// TIA Portal project "KNX_SPS_Forum_Van" (V18)

(* hardware
DEVICE "S7-1200-Station_1"  S7-1200 Station
   slot 0: "Baugruppenträger_0"  S7-1200 Rack  Rack  V1.0
   slot 1: "PLC_1"  CPU 1214C DC/DC/DC  6ES7 214-1AG40-0XB0  V4.6
*)

// ===== PLC "PLC_1"  CPU 1214C DC/DC/DC =====

VAR_GLOBAL CONSTANT   // PLC tag table "CONST_KNX"
   "KNX_ARRAY_MAX" : Int := 49;
END_VAR

VAR_GLOBAL CONSTANT   // PLC tag table "CONST_Ethernet"
   "CONN_ID_KNX" : Int := 1;
   "CONN_ID_SMA" : Conn_Ouc := 2;
   "CONN_ID_RASENROBI" : Conn_Ouc := 3;
   "CONN_ID_VOLKSZAEHLER_GET" : Conn_Ouc := 4;
   "CONN_ID_SHELLY" : Conn_Ouc := 5;
   "CONN_ID_VOLKSZAEHLER_POST" : Conn_Ouc := 6;
   "CONN_ID_WALLBOX" : Conn_Ouc := 7;
   "CONN_ID_Res8" : Conn_Ouc := 8;
   "Maximal 8 OU Verbindungen" : Conn_Ouc := 8888;   // Maximal 8 OU Verbindungen
END_VAR

// folder: KNX

TYPE "KNX_Data_Exchange"
   STRUCT
      Empf_Dat : "KNX_Empf_Dat";
      Send_Dat : "KNX_Send_Dat";
      Senden : Bool;
      Empfangen : Bool;
   END_STRUCT;
   // // Empf_Dat.Daten[1] : APCI + 6Bit Nutzdaten
END_TYPE

TYPE "KNX_Empf_Dat"
   STRUCT
      GruppenAddr : Word;
      Laenge : Byte;
      NPDU_ABCI : Byte;
      Daten : Array[1..20] of Byte;
   END_STRUCT;
END_TYPE

TYPE "KNX_Send_Dat"
   STRUCT
      GruppenAddr : Word;
      Laenge : Byte;
      NPDU_ABCI : Byte;
      Daten : Array[1..20] of Byte;
   END_STRUCT;
END_TYPE

TYPE "KNX_Data_Exchange_bak"
   STRUCT
      Empf_Dat : Struct
         GruppenAddr : Word;
         Laenge : Byte;
         NPDU_ABCI : Byte;
         Daten : Array[1..20] of Byte;
      END_STRUCT;
      Send_Dat : Struct
         GruppenAddr : Word;
         Laenge : Byte;
         NPDU_ABCI : Byte;
         Daten : Array[1..20] of Byte;
      END_STRUCT;
      Senden : Bool;
      Empfangen : Bool;
   END_STRUCT;
END_TYPE

TYPE "KNX_GA_Nr"
   STRUCT
      haupt : USInt;   // Hauptgruppe = 0..31
      mittel : USInt;   // Mittelgruppe = 0..7
      unter : USInt;   // Untergruppe = 0..255
   END_STRUCT;
END_TYPE

TYPE "KNX_Log_empf"
   STRUCT
      ga_nr : "KNX_GA_Nr";
      Empf_Dat : "KNX_Empf_Dat";
   END_STRUCT;
END_TYPE

TYPE "KNX_test_2"
   STRUCT
      GA : "KNX_GA_Nr";
      para : Struct
         aktiv : Bool;
         abfragbar : Bool;   // ReadRequest vom(!) Bus beantworten
         beschreibbar : Bool;   // Write vom(!) Bus zulassen
         initScan : Bool;   // ist diese Option aktiviert wird der KO-Wert beim Start vom KNX-Bus abgefragt (Read-Request)
         sendByChange : Bool;
         sendByChangeValue : Real;
      END_STRUCT;
      cmd : Struct
         send : Bool;   // SPS Wert an den Bus senden
         sendReadRequest : Bool;   // Wert vom Bus abfragen
      END_STRUCT;
      value : Struct
         DPT : UInt;
         DPT1 : Bool;
         DPT2 : Byte;
         DPT3 : Byte;
         DPT4 : Char;
         DPT5 : USInt;
         DPT6 : SInt;
         DPT7 : UInt;
         DPT8 : Int;
         DPT9 : Real;
         DPT10x : Bool;
         DPT11x : Bool;
         DPT12 : UDInt;
         DPT13 : DInt;
         DPT14 : Real;
      END_STRUCT;
   END_STRUCT;
END_TYPE

TYPE "KNX_test_1"
   STRUCT
      GA : "KNX_GA_Nr";
      para : Struct
         aktiv : Bool;
         abfragbar : Bool;   // ReadRequest vom(!) Bus beantworten
         beschreibbar : Bool;   // Write vom(!) Bus zulassen
         initScan : Bool;   // ist diese Option aktiviert wird der KO-Wert beim Start vom KNX-Bus abgefragt (Read-Request)
         sendByChange : Bool;
         sendByChangeValue : Real;
      END_STRUCT;
      cmd : Struct
         send : Bool;   // SPS Wert an den Bus senden
         sendReadRequest : Bool;   // Wert vom Bus abfragen
      END_STRUCT;
      value : Struct
         DPT : Int;
         raw : Array[0..14] of Byte;
      END_STRUCT;
   END_STRUCT;
END_TYPE

TYPE "KNX_KO"
   STRUCT
      GA : "KNX_GA_Nr";   // Gruppenadresse
      para : Struct   // Parameter
         aktiv : Bool;   // KO ist aktiv und wird bearbeitet
         abfragbarVomBus : Bool;   // SPS Sendet Wert auf den Bus - ReadRequest vom(!) Bus beantworten
         beschreibbarVomBus : Bool;   // SPS empfängt Wert vom Bus - Write vom(!) Bus zulassen
         initScan : Bool;   // ist diese Option aktiviert wird der KO-Wert beim Start vom KNX-Bus abgefragt (Read-Request)
         sendByChange : Bool;   // Auf den Bus senden wenn sich der SPS Wert geändert hat
         sendByChangeValue : Real;   // diffferenz um den sich der Wert ändern muss
      END_STRUCT;
      cmd : Struct   // Kommando
         send : Bool;   // SPS Wert an den Bus senden
         readRequest : Bool;   // Wert vom Bus abfragen
      END_STRUCT;
      stat : Struct   // Status
         newTelegramRec : Bool;   // Neues Telegram empfangen
         newTelegramSend : Bool;   // Telegram gesendet
         counterRec : UInt;   // Zähler Telegramme Empfangen (Flanke)
         counterSend : UInt;   // Zähler Telegramme Gesendet
      END_STRUCT;
   END_STRUCT;
END_TYPE

TYPE "KNX_DPT3"
   STRUCT
      Down_Increase : Bool;   // 0 = Up, Decrease / 1 = Down, Increase
      prozent : USInt;   // 1, 3, 6, 12, 25, 50, 100% / 0 = Stopp
   END_STRUCT;
END_TYPE

// folder: 10 Haus Logik/instanzen

DATA_BLOCK "aussen-rasenrobi_DB"   // DB8
{ S7_Optimized_Access := 'TRUE' }
VERSION : 0.1
// stored: InstanceOfName aussen-rasenrobi
"aussen-rasenrobi"
BEGIN
END_DATA_BLOCK

DATA_BLOCK "eg-Wohn-Ess-Kueche_DB"   // DB17
{ S7_Optimized_Access := 'TRUE' }
VERSION : 0.1
// stored: InstanceOfName eg-Wohn-Ess-Kueche
"eg-Wohn-Ess-Kueche"
BEGIN
END_DATA_BLOCK

DATA_BLOCK "zental-strom_DB"   // DB21
{ S7_Optimized_Access := 'TRUE' }
VERSION : 0.1
// stored: InstanceOfName zental-strom
"zental-strom"
BEGIN
END_DATA_BLOCK

DATA_BLOCK "zentral-wasser_DB"   // DB33
{ S7_Optimized_Access := 'TRUE' }
VERSION : 0.1
// stored: InstanceOfName zentral-wasser
"zentral-wasser"
BEGIN
END_DATA_BLOCK

DATA_BLOCK "zentral-beschattung_DB"   // DB35
{ S7_Optimized_Access := 'TRUE' }
VERSION : 0.1
// stored: InstanceOfName zentral-beschattung
"zentral-beschattung"
BEGIN
END_DATA_BLOCK

// folder: 20 KNX

DATA_BLOCK "db-knx-Allg"   // DB2
{ S7_Optimized_Access := 'TRUE' }
VERSION : 0.1
   VAR
      "Disconnect Count" : Int;
      DisconnectChannelID : Array[1..20] of Byte;
      knxComOk : Bool;
      knxComTimeOut : Bool;
      initScanDone : Bool;
      knxBereit : Bool;
   END_VAR
BEGIN
END_DATA_BLOCK

DATA_BLOCK "db-knx-log"   // DB4
{ S7_Optimized_Access := 'TRUE' }
VERSION : 0.1
   VAR
      index : Int;
      empf : Array[0..100] of "KNX_Log_empf";
   END_VAR
BEGIN
END_DATA_BLOCK

DATA_BLOCK "db-knx-com"   // DB10
{ S7_Optimized_Access := 'TRUE' }
VERSION : 0.1
   VAR
      KNXDat : "KNX_Data_Exchange";   // KNX: Datenaustausch zwischen den FBs
   END_VAR
BEGIN
END_DATA_BLOCK

DATA_BLOCK "db-knx-ko"   // DB15
{ S7_Optimized_Access := 'TRUE' }
VERSION : 0.1
   VAR
      ko : Array[0.."KNX_ARRAY_MAX"] of "KNX_KO";   // Kommunikationsobjekt
      koVal : Struct   // Kommunikationsobjekt Wert
         "0_Terassen-Tür (Zu=Aus=0 / Auf=Ein=1)" : Bool;   // 6/1/2 = Terassen-Tür (Zu=Aus=0 / Auf=Ein=1)
         "1_Wohn-Ess-Kueche.Terasse(Patch-kurz)" : Bool;   // 6/1/6 = Wohn-Ess-Kueche.Terasse(Patch-kurz)
         "2_Wohn-Ess-Küche.Szene" : USInt;   // 8/1/1 = Wohn-Ess-Küche.Szene
         "3_Wohnen-Tür-SW.Jal(Jalousie Auf/Ab)" : Bool;   // 3/1/140 = Wohnen-Tür-SW.Jal(Jalousie Auf/Ab)
         "4_Zisterne(Fuellstand qm)" : Real;   // 6/3/140 = Zisterne(Fuellstand qm)
         "5_PV-Anlage(Erzeugung)" : Real;   // 6/3/141 = PV-Anlage(Erzeugung) / DPT 9.024 Leistung (kW)
         "6_Stromzaehler(In-Out-Aktuell)" : Real;   // 6/0/0 = Stromzaehler(In-Out-Aktuell) / Positiv=Bezug vom Netz / Negativ = Verkauf an Netz / / DPT 9.024 Leistung (kW)
         "7_Strom(Eigenverbrauch)" : Real;   // 6/0/1 = Strom(Eigenverbrauch) / DPT 9.024 Leistung (kW)
         "8_Zirkulation.WarmWasser(Ein)" : Bool;   // 7/0/1 = Zirkulation.WarmWasser(Ein)
         "9_Umwelt.Wetterstation(Helligkeit O Messwert)" : Real;   // 6/3/0 = Umwelt.Wetterstation(Helligkeit O Messwert)
         "10_Umwelt.Wetterstation(Helligkeit S Messwert)" : Real;   // 6/3/17 = Umwelt.Wetterstation(Helligkeit S Messwert)
         "11_Umwelt.Wetterstation(Helligkeit W Messwert)" : Real;   // 6/3/34 = Umwelt.Wetterstation(Helligkeit W Messwert)
         "12_Umwelt-Garage.Lichtsensor(Helligkeit Messwert)" : Real;   // 6/3/105 = Umwelt-Garage.Lichtsensor(Helligkeit Messwert)
         "13_Beschattung(Diag)" : String[14];   // 3/1/221 = Beschattung(Diag)
         "14_Umwelt.Wetterstation(Wind Geschwindigkeit)" : Real;   // 6/3/54 = Umwelt.Wetterstation(Wind Geschwindigkeit)
         "15_Umwelt.Wetterstation(Temperatur Messwert)" : Real;   // 6/3/55 = Umwelt.Wetterstation(Temperatur Messwert)
         "16_Umwelt.Helligkeit.Max(Helligkeit)" : Real;   // 6/3/106 = Umwelt.Helligkeit.Max(Helligkeit)
         "17_Umwelt.Regensensor(Meldung Regen ja/nein)" : Bool;   // 6/3/100 = Umwelt.Regensensor(Meldung Regen ja/nein)
         "18_DPT3_Test" : "KNX_DPT3";   // 11/0/10 = DPT3 Test
      END_STRUCT;
   END_VAR
   VAR RETAIN
      initScan_nachDbReinit : Bool := false;   // Löst einen InitScan aus nachdem der DB reinitialisiert wurde
   END_VAR
BEGIN
   ko[0].GA.haupt := 6;
   ko[0].GA.mittel := 1;
   ko[0].GA.unter := 2;
   ko[0].para.aktiv := true;
   ko[0].para.abfragbarVomBus := false;
   ko[0].para.beschreibbarVomBus := true;
   ko[0].para.initScan := true;
   ko[1].GA.haupt := 6;
   ko[1].GA.mittel := 1;
   ko[1].GA.unter := 6;
   ko[1].para.aktiv := true;
   ko[1].para.abfragbarVomBus := false;
   ko[1].para.beschreibbarVomBus := true;
   ko[1].para.initScan := false;
   ko[1].para.sendByChange := false;
   ko[2].GA.haupt := 8;
   ko[2].GA.mittel := 1;
   ko[2].GA.unter := 1;
   ko[2].para.aktiv := true;
   ko[2].para.abfragbarVomBus := false;
   ko[2].para.beschreibbarVomBus := true;
   ko[2].para.initScan := false;
   ko[2].para.sendByChange := false;
   ko[3].GA.haupt := 3;
   ko[3].GA.mittel := 1;
   ko[3].GA.unter := 140;
   ko[3].para.aktiv := true;
   ko[3].para.abfragbarVomBus := false;
   ko[3].para.beschreibbarVomBus := false;
   ko[3].para.initScan := false;
   ko[4].GA.haupt := 6;
   ko[4].GA.mittel := 3;
   ko[4].GA.unter := 140;
   ko[4].para.aktiv := true;
   ko[4].para.abfragbarVomBus := true;
   ko[4].para.beschreibbarVomBus := false;
   ko[4].para.initScan := false;
   ko[4].para.sendByChange := true;
   ko[4].para.sendByChangeValue := 0.05;
   ko[5].GA.haupt := 6;
   ko[5].GA.mittel := 3;
   ko[5].GA.unter := 141;
   ko[5].para.aktiv := true;
   ko[5].para.abfragbarVomBus := true;
   ko[5].para.beschreibbarVomBus := false;
   ko[5].para.initScan := false;
   ko[5].para.sendByChange := true;
   ko[5].para.sendByChangeValue := 0.2;
   ko[6].GA.haupt := 6;
   ko[6].GA.unter := 0;
   ko[6].para.aktiv := true;
   ko[6].para.initScan := false;
   ko[7].GA.haupt := 6;
   ko[7].GA.mittel := 0;
   ko[7].GA.unter := 1;
   ko[7].para.aktiv := true;
   ko[7].para.initScan := false;
   ko[8].GA.haupt := 7;
   ko[8].GA.unter := 1;
   ko[8].para.aktiv := true;
   ko[8].GA.mittel := 0;
   ko[6].GA.mittel := 0;
   ko[6].para.abfragbarVomBus := true;
   ko[6].para.beschreibbarVomBus := false;
   ko[6].para.sendByChange := true;
   ko[6].para.sendByChangeValue := 0.2;
   ko[7].para.abfragbarVomBus := true;
   ko[7].para.beschreibbarVomBus := false;
   ko[7].para.sendByChange := true;
   ko[7].para.sendByChangeValue := 0.2;
   ko[9].GA.haupt := 6;
   ko[9].GA.mittel := 3;
   ko[9].GA.unter := 0;
   ko[9].para.aktiv := true;
   ko[9].para.abfragbarVomBus := false;
   ko[9].para.initScan := true;
   ko[9].para.beschreibbarVomBus := true;
   ko[9].para.sendByChange := false;
   ko[10].GA.haupt := 6;
   ko[10].GA.mittel := 3;
   ko[10].GA.unter := 17;
   ko[10].para.aktiv := true;
   ko[10].para.abfragbarVomBus := false;
   ko[10].para.beschreibbarVomBus := true;
   ko[10].para.initScan := true;
   ko[10].para.sendByChange := false;
   ko[11].GA.haupt := 6;
   ko[11].GA.mittel := 3;
   ko[11].GA.unter := 34;
   ko[11].para.aktiv := true;
   ko[11].para.abfragbarVomBus := false;
   ko[11].para.beschreibbarVomBus := true;
   ko[11].para.initScan := true;
   ko[11].para.sendByChange := false;
   ko[12].GA.haupt := 6;
   ko[12].GA.mittel := 3;
   ko[12].GA.unter := 105;
   ko[12].para.aktiv := true;
   ko[12].para.abfragbarVomBus := false;
   ko[12].para.beschreibbarVomBus := true;
   ko[12].para.initScan := true;
   ko[12].para.sendByChange := false;
   ko[13].GA.haupt := 3;
   ko[13].GA.mittel := 1;
   ko[13].GA.unter := 221;
   ko[13].para.aktiv := true;
   ko[13].para.abfragbarVomBus := false;
   ko[13].para.beschreibbarVomBus := true;
   ko[13].para.initScan := true;
   ko[13].para.sendByChange := false;
   ko[14].GA.haupt := 6;
   ko[14].GA.mittel := 3;
   ko[14].GA.unter := 54;
   ko[14].para.aktiv := true;
   ko[14].para.abfragbarVomBus := false;
   ko[14].para.beschreibbarVomBus := true;
   ko[14].para.initScan := true;
   ko[14].para.sendByChange := false;
   ko[15].GA.haupt := 6;
   ko[15].GA.mittel := 3;
   ko[15].GA.unter := 55;
   ko[15].para.aktiv := true;
   ko[15].para.abfragbarVomBus := false;
   ko[15].para.beschreibbarVomBus := true;
   ko[15].para.initScan := true;
   ko[15].para.sendByChange := false;
   ko[16].GA.haupt := 6;
   ko[16].GA.mittel := 3;
   ko[16].GA.unter := 106;
   ko[16].para.aktiv := true;
   ko[16].para.abfragbarVomBus := true;
   ko[16].para.beschreibbarVomBus := false;
   ko[16].para.initScan := false;
   ko[16].para.sendByChange := true;
   ko[16].para.sendByChangeValue := 100.0;
   ko[17].GA.haupt := 6;
   ko[17].GA.mittel := 3;
   ko[17].GA.unter := 100;
   ko[17].para.aktiv := true;
   ko[17].para.initScan := true;
   ko[17].para.beschreibbarVomBus := true;
   ko[18].GA.haupt := 11;
   ko[18].GA.mittel := 0;
   ko[18].GA.unter := 10;
   ko[18].para.aktiv := true;
   ko[18].para.abfragbarVomBus := true;
   ko[18].para.beschreibbarVomBus := true;
   ko[18].para.initScan := true;
   ko[18].para.sendByChange := true;
   // ko[0] : 6/1/2 = Terassen-Tür (Zu=Aus=0 / Auf=Ein=1)
   // ko[1] : 6/1/6 = Wohn-Ess-Kueche.Terasse(Patch-kurz)
   // ko[2] : 8/1/1 = Wohn-Ess-Küche.Szene
   // ko[3] : 3/1/140 = Wohnen-Tür-SW.Jal(Jalousie Auf/Ab)
   // ko[4] : 6/3/140 = Zisterne(Fuellstand qm)
   // ko[5] : 6/3/141 = PV-Anlage(Erzeugung)
   // ko[6] : 6/0/0 = Stromzaehler(In-Out-Aktuell)
   // ko[7] : 6/0/1 = Strom(Eigenverbrauch)
   // ko[8] : 7/0/1 = Zirkulation.WarmWasser(Ein)
   // ko[9] : 6/3/0 = Umwelt.Wetterstation(Helligkeit O Messwert)
   // ko[10] : 6/3/17 = Umwelt.Wetterstation(Helligkeit S Messwert)
   // ko[11] : 6/3/34 = Umwelt.Wetterstation(Helligkeit W Messwert)
   // ko[12] : 6/3/105 = Umwelt-Garage.Lichtsensor(Helligkeit Messwert)
   // ko[13] : 3/1/221 = Beschattung(Diag)
   // ko[14] : 6/3/54 = Umwelt.Wetterstation(Wind Geschwindigkeit)
   // ko[15] : 6/3/55 = Umwelt.Wetterstation(Temperatur Messwert)
   // ko[16] : 6/3/106 = Umwelt.Helligkeit.Max(Helligkeit)
   // ko[17] : 6/3/100 = Umwelt.Regensensor(Meldung Regen ja/nein)
   // ko[18] : 11/0/10 = DPT3 Test
END_DATA_BLOCK

// folder: 20 KNX/instanzen

DATA_BLOCK "KNX_Kommunikation_DB"   // DB1
{ S7_Optimized_Access := 'TRUE' }
VERSION : 0.1
// stored: InstanceOfName KNX_Kommunikation
"KNX_Kommunikation"
BEGIN
END_DATA_BLOCK

DATA_BLOCK "knx-ko-aufrufe_DB"   // DB3
{ S7_Optimized_Access := 'TRUE' }
VERSION : 0.1
// stored: InstanceOfName knx-ko-aufrufe
"knx-ko-aufrufe"
BEGIN
END_DATA_BLOCK

DATA_BLOCK "knx-com_DB"   // DB11
{ S7_Optimized_Access := 'TRUE' }
VERSION : 0.1
// stored: InstanceOfName knx-com
"knx-com"
BEGIN
END_DATA_BLOCK

// folder: (top level)

ORGANIZATION_BLOCK "Main"   // OB1, SCL, ProgramCycle
TITLE = "Main Program Sweep (Cycle)"
{ S7_Optimized_Access := 'TRUE' }
VERSION : 0.1
   VAR_INPUT
      Initial_Call : Bool;   // Initial call of this OB
      Remanence : Bool;   // =True, if remanent data are available
   END_VAR
BEGIN


   // Haus Logik
   "zental-strom_DB"();
   "zentral-wasser_DB"();
   "zentral-beschattung_DB"();

   "eg-Wohn-Ess-Kueche_DB"();

   "aussen-rasenrobi_DB"();




   // KNX Kommunikation
   "knx-com_DB"();
   "knx-ko-aufrufe_DB"();
END_ORGANIZATION_BLOCK

// folder: 10 Haus Logik/0 Zentral

FUNCTION_BLOCK "zental-strom"   // FB23, FBD
TITLE = Strom
{ S7_Optimized_Access := 'TRUE' }
VERSION : 0.1
BEGIN

REGION Network 1 (SCL): Eigenverbrauch / PV Überschuss
   // "db-knx-ko".koVal."6_Stromzaehler(In-Out-Aktuell)"
   // "db-knx-ko".koVal."5_PV-Anlage(Erzeugung)"

   // Netz
   // Positiv : Strom Bezug vom Netz
   // Negativ : Strom Verkauf an Netz

   //"db-knx-ko".koVal."7_Strom(Eigenverbrauch)" := ("db-knx-ko".koVal."5_PV-Anlage(Erzeugung)" + "db-knx-ko".koVal."6_Stromzaehler(In-Out-Aktuell)");

   "db-haus".strom.eigenverbrauch_W := ("db-haus".strom.pv_W + "db-haus".strom.netz_W);
   "db-haus".strom.eigenverbrauchOhneWB_W := ("db-haus".strom.eigenverbrauch_W - "db-haus".strom.wallbox_W);



   "db-haus".strom.pvUeberschuss_W := ("db-haus".strom.netz_W * -1.0);

   //"db-haus".strom.pvUeberschussOhneWB_W := ("db-haus".strom.pvUeberschuss_W - "db-haus".strom.wallbox_W);

   "db-haus".strom.pvUeberschussOhneWB_W := "db-haus".strom.pv_W - "db-haus".strom.eigenverbrauchOhneWB_W;
END_REGION
END_FUNCTION_BLOCK

FUNCTION_BLOCK "zentral-wasser"   // FB28, FBD
TITLE = Zentral - Wasser
{ S7_Optimized_Access := 'TRUE' }
VERSION : 0.1
   VAR
      sperre : TOF_TIME;
   END_VAR
   VAR_TEMP   // added for the SCL form of the ladder/FBD networks
      _w1 : Bool;
      _w2 : Bool;
   END_VAR
BEGIN

REGION Network 1: Zirkulationspumpe
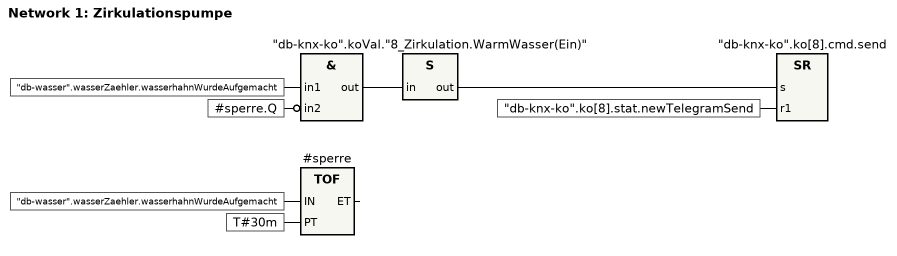
   #_w1 := "db-wasser".wasserZaehler.wasserhahnWurdeAufgemacht AND NOT #sperre.Q;
   IF #_w1 THEN "db-knx-ko".koVal."8_Zirkulation.WarmWasser(Ein)" := TRUE; END_IF;
   #_w2 := "db-knx-ko".ko[8].stat.newTelegramSend;
   IF #_w1 THEN
       "db-knx-ko".ko[8].cmd.send := TRUE;   // SR flip-flop
   END_IF;
   IF #_w2 THEN "db-knx-ko".ko[8].cmd.send := FALSE; END_IF;
   #sperre(IN := "db-wasser".wasserZaehler.wasserhahnWurdeAufgemacht, PT := T#30m);   // TOF
END_REGION
END_FUNCTION_BLOCK

FUNCTION_BLOCK "zentral-beschattung"   // FB31, FBD
{ S7_Optimized_Access := 'TRUE' }
VERSION : 0.1
   VAR_TEMP
      helligkeitGarage : Real;
   END_VAR
BEGIN

REGION Network 1 (SCL): Sonnenstand - Diagnoseobjekt de Jal-Aktors - INFO
   (*

   Diagnoseobjekt de Jal-Aktors

   Diagnoseobjekt 
   Das Diagnoseobjekt kann als Status für Visualisierungen oder zur Inbetriebnahme/Diagnose 
   verwendet werden. Es enthält Informationen zur Bereitschaft der Beschattung, Schwellwert, Azimut 
   und Elevation (siehe hierzu auch 4.13.3 Grundlagen der Sonnenstands Berechnung) aus. Das 
   Diagnoseobjekt ist dabei wie folgt aufgebaut: 
   M1 S1 A150 E30 
    Mx 
   Anzeige des Beschattungsmodus; bit-codiert: 
    Bit 1: 0 = Beschattung nicht bereit, 1 = Beschattung bereit 
    Bit 2: 0 = Beschattung nicht gesperrt, 1 = Beschattung gesperrt 
    Bit 3: 0 = keine Außentemperatursperre, 1 = Außentemperatursperre aktiv 
   Bsp: M6-> in binärer Form: 110 -> Beschattung gesperrt und Temperatursperre aktiv 



    Sx 
   Anzeige ob Schwelle 1/2 überschritten ist 
    S0: keine Schwelle ist überschritten 
    S1: Helligkeitsschwelle 1 ist überschritten 
    S2: Helligkeitsschwelle 2 ist überschritten 
    Axxx 
   Ausgabe des Azimuts (Sonnenwinkel) der Sonne in Grad 
    Exx 
   Ausgabe der Elevation (Sonnenhöhe) der Sonne in Grad 
   Kommt die Meldung ERR: Date, so wurde kein Wert für Datum/Uhrzeit empfangen. 
   *)
END_REGION

REGION Network 2 (SCL): Sonnenstand - Aufschlüsseln

   // 12345678901111
   //          11234
   // M1 S1 A150 E30

   "db-haus".besch.sonnenstand.azimut := STRING_TO_REAL(MID(IN:="db-knx-ko".koVal."13_Beschattung(Diag)", L:=3, P:=8));
   "db-haus".besch.sonnenstand.elevation := STRING_TO_REAL(MID(IN := "db-knx-ko".koVal."13_Beschattung(Diag)", L := 2, P := 13));
END_REGION

REGION Network 3: Maximaler Helligkeitswert
   // Im Sommer kann es passieren das bei hohem Sonnenstand der Dachvorsprung die Wetterstation verschattet, und somit die Beschattung aus geht.
   // Jetzt soll der Sensor auf der Garage einnen besseren Helligkeitswert liefern
   // 
   // Helligkeitsensor der Garage nur Berücksichtigen wenn Beschattung an Hausfront SW aktiv (Azimut zwischen 160-270°)
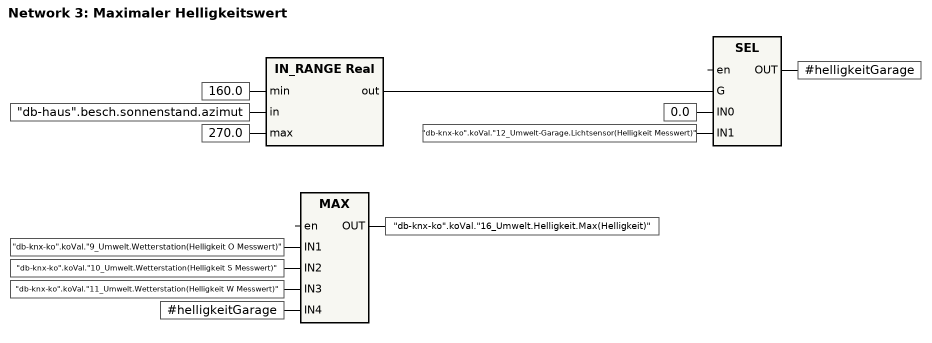
   #helligkeitGarage := SEL(G := (160.0 <= "db-haus".besch.sonnenstand.azimut) AND ("db-haus".besch.sonnenstand.azimut <= 270.0), IN0 := 0.0, IN1 := "db-knx-ko".koVal."12_Umwelt-Garage.Lichtsensor(Helligkeit Messwert)");
   "db-knx-ko".koVal."16_Umwelt.Helligkeit.Max(Helligkeit)" := MAX(IN1 := "db-knx-ko".koVal."9_Umwelt.Wetterstation(Helligkeit O Messwert)", IN2 := "db-knx-ko".koVal."10_Umwelt.Wetterstation(Helligkeit S Messwert)", IN3 := "db-knx-ko".koVal."11_Umwelt.Wetterstation(Helligkeit W Messwert)", IN4 := #helligkeitGarage);
END_REGION
END_FUNCTION_BLOCK

// folder: 10 Haus Logik/1 EG

FUNCTION_BLOCK "eg-Wohn-Ess-Kueche"   // FB17, FBD
{ S7_Optimized_Access := 'TRUE' }
VERSION : 0.1
   VAR_TEMP   // added for the SCL form of the ladder/FBD networks
      _w1 : Bool;
      _w2 : Bool;
      _w3 : Bool;
      _w4 : Bool;
      _w5 : Bool;
   END_VAR
BEGIN

REGION Network 1: Patch Taste neben der Terassentür
   // Tür Offen  -> Jal an der Tür Auf   -> Wohnen-Tür-SW.Jal(Jalousie Auf/Ab)  AUF
   // Tür Zu       -> Alle Jal Auf              -> Szene 1 (0)
   // 
   // 1.008 DPT_UpDown 0 = Up / 1 = Down 
   // Szene auf dem Bus immer -1 (null Index)
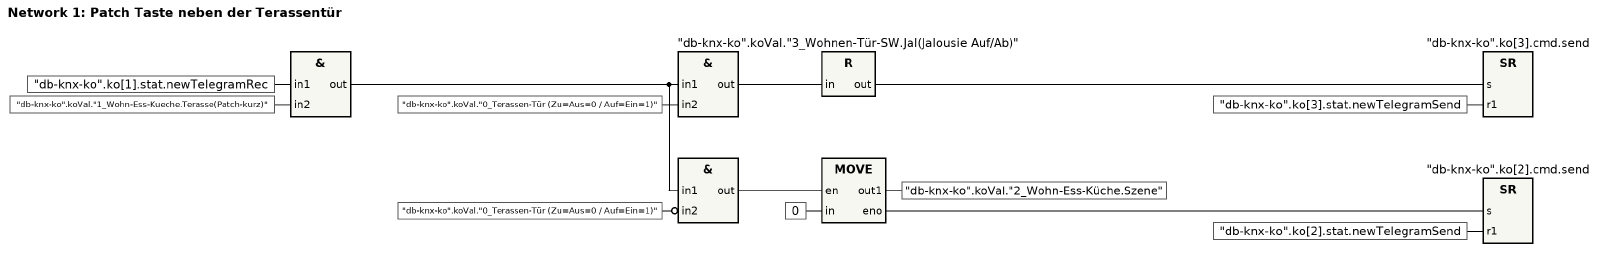
   #_w1 := "db-knx-ko".ko[1].stat.newTelegramRec AND "db-knx-ko".koVal."1_Wohn-Ess-Kueche.Terasse(Patch-kurz)";
   #_w2 := #_w1 AND "db-knx-ko".koVal."0_Terassen-Tür (Zu=Aus=0 / Auf=Ein=1)";
   IF #_w2 THEN "db-knx-ko".koVal."3_Wohnen-Tür-SW.Jal(Jalousie Auf/Ab)" := FALSE; END_IF;
   #_w3 := "db-knx-ko".ko[3].stat.newTelegramSend;
   IF #_w2 THEN
       "db-knx-ko".ko[3].cmd.send := TRUE;   // SR flip-flop
   END_IF;
   IF #_w3 THEN "db-knx-ko".ko[3].cmd.send := FALSE; END_IF;
   #_w4 := #_w1 AND NOT "db-knx-ko".koVal."0_Terassen-Tür (Zu=Aus=0 / Auf=Ein=1)";
   IF #_w4 THEN "db-knx-ko".koVal."2_Wohn-Ess-Küche.Szene" := 0; END_IF;
   #_w5 := "db-knx-ko".ko[2].stat.newTelegramSend;
   IF #_w4 THEN
       "db-knx-ko".ko[2].cmd.send := TRUE;   // SR flip-flop
   END_IF;
   IF #_w5 THEN "db-knx-ko".ko[2].cmd.send := FALSE; END_IF;
END_REGION

REGION Network 2 (SCL): Szenen Info
   (*

   Die "Technische" Szenen Nummer ist immer -1 zu der in der ETS angezeigten/parametrierten Nummer

    DPT_SceneControl allows numbering the scene from 0 to 63. KNX Association recommends displaying these scene 
   numbers in ETS™, other software and controllers numbered from 1 to 64, this is, with an offset of 1 compared to the actual 
   transmitted value. 

   *)
END_REGION
END_FUNCTION_BLOCK

// folder: 10 Haus Logik/3 Aussen

FUNCTION_BLOCK "aussen-rasenrobi"   // FB2, FBD
TITLE = Aussen - Rasen Roboter
{ S7_Optimized_Access := 'TRUE' }
VERSION : 0.1
   VAR
      TOF_Regen : TOF_TIME;
      TOF_Windalarm : TOF_TIME;
      TON_Regendauer : TON_TIME;
      fl_regenEnde : Bool;
      TON_Tempalarm : TON_TIME;
   END_VAR
   VAR_TEMP   // added for the SCL form of the ladder/FBD networks
      _w1 : Bool;
   END_VAR
BEGIN

REGION Network 1: Regendauer erfassen
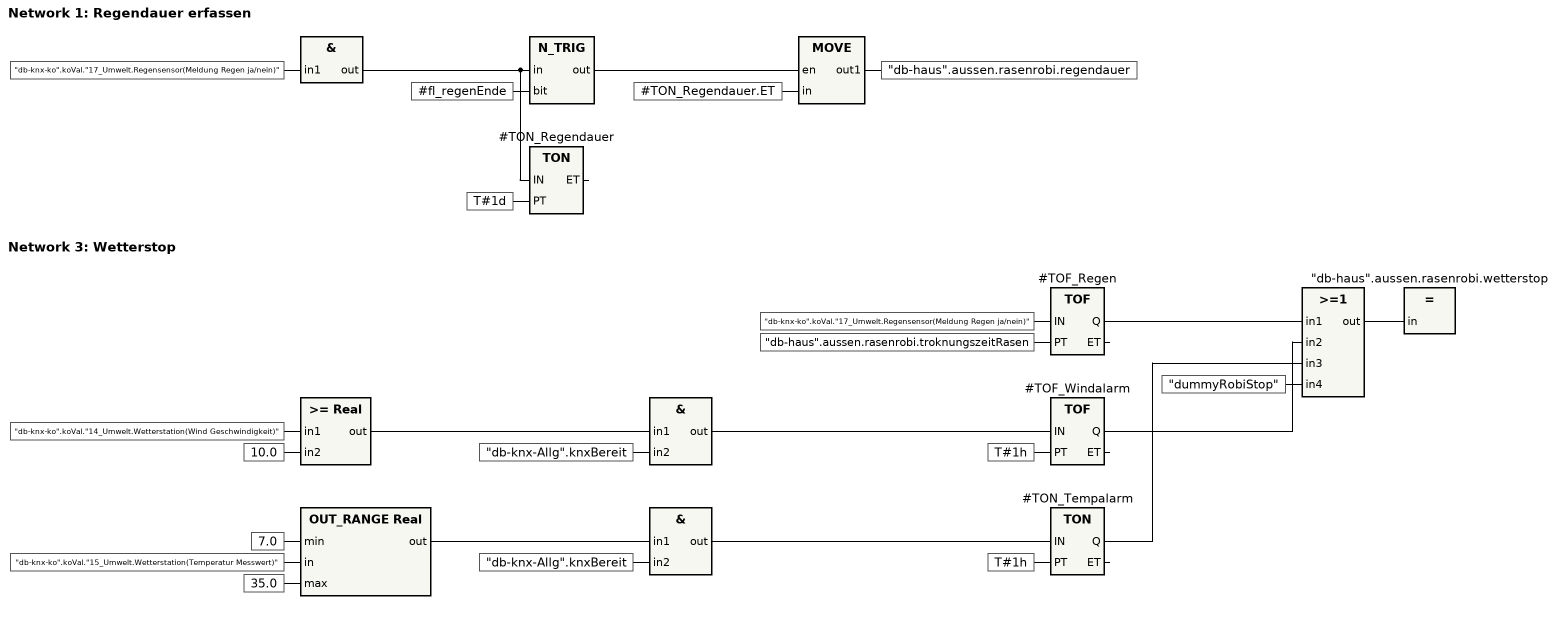
   #_w1 := NOT "db-knx-ko".koVal."17_Umwelt.Regensensor(Meldung Regen ja/nein)" AND #fl_regenEnde;   // falling edge
   #fl_regenEnde := "db-knx-ko".koVal."17_Umwelt.Regensensor(Meldung Regen ja/nein)";
   IF #_w1 THEN "db-haus".aussen.rasenrobi.regendauer := #TON_Regendauer.ET; END_IF;
   #TON_Regendauer(IN := "db-knx-ko".koVal."17_Umwelt.Regensensor(Meldung Regen ja/nein)", PT := T#1d);   // TON
END_REGION

REGION Network 2 (SCL): Troknungszeit des Rasens
   // Je länger es geregnet hat, desto länger soll die Troknungszeit des Rasens sein

   "db-haus".aussen.rasenrobi.troknungszeitRasen := t#1h + REAL_TO_DINT((DINT_TO_REAL(TIME_TO_DINT("db-haus".aussen.rasenrobi.regendauer)) * 0.1));
END_REGION

REGION Network 3: Wetterstop
   #TOF_Regen(IN := "db-knx-ko".koVal."17_Umwelt.Regensensor(Meldung Regen ja/nein)",   // TOF
              PT := "db-haus".aussen.rasenrobi.troknungszeitRasen);
   #TOF_Windalarm(IN := ("db-knx-ko".koVal."14_Umwelt.Wetterstation(Wind Geschwindigkeit)" >= 10.0) AND "db-knx-Allg".knxBereit,   // TOF
                  PT := T#1h);
   #TON_Tempalarm(IN := (("db-knx-ko".koVal."15_Umwelt.Wetterstation(Temperatur Messwert)" < 7.0) OR ("db-knx-ko".koVal."15_Umwelt.Wetterstation(Temperatur Messwert)" > 35.0)) AND "db-knx-Allg".knxBereit,   // TON
                  PT := T#1h);
   "db-haus".aussen.rasenrobi.wetterstop := #TOF_Regen.Q OR #TOF_Windalarm.Q OR #TON_Tempalarm.Q OR "dummyRobiStop";
END_REGION
END_FUNCTION_BLOCK

// folder: 20 KNX

FUNCTION_BLOCK "knx-ko-aufrufe"   // FB10, FBD
{ S7_Optimized_Access := 'TRUE' }
VERSION : 0.1
   VAR
      "knx-KO" : Array[0.."KNX_ARRAY_MAX"] of "knx-KO";
   END_VAR
BEGIN

REGION Network 1 (SCL): INFO
   (*

   Im Datenbaustein "db-knx-ko" müssen die KOs (Kommunikationsobjekte) entsprechend angelegt und konfiguriert werden.
   Und dann hier aufgerufen werden

   *)
END_REGION

REGION Network 2 (SCL): Terassen-Tür / Jalllosie


   // 6/1/6 = Wohn-Ess-Kueche.Terasse(Patch-kurz)
   #"knx-KO"[1](Wert := "db-knx-ko".koVal."1_Wohn-Ess-Kueche.Terasse(Patch-kurz)",
                KNX_KO := "db-knx-ko".ko[1],
                KNX_Dat := "db-knx-com".KNXDat);

   // 6/1/2 = Terassen-Tür (Zu=Aus=0 / Auf=Ein=1)
   #"knx-KO"[0](Wert := "db-knx-ko".koVal."0_Terassen-Tür (Zu=Aus=0 / Auf=Ein=1)",
                KNX_KO := "db-knx-ko".ko[0],
                KNX_Dat := "db-knx-com".KNXDat);




   // 8/1/1 = Wohn-Ess-Küche.Szene
   #"knx-KO"[2](Wert := "db-knx-ko".koVal."2_Wohn-Ess-Küche.Szene", KNX_KO := "db-knx-ko".ko[2], KNX_Dat := "db-knx-com".KNXDat);

   // 3/1/140 = Wohnen-Tür-SW.Jal(Jalousie Auf/Ab)
   #"knx-KO"[3](Wert := "db-knx-ko".koVal."3_Wohnen-Tür-SW.Jal(Jalousie Auf/Ab)",
                KNX_KO := "db-knx-ko".ko[3],
                KNX_Dat := "db-knx-com".KNXDat);
END_REGION

REGION Network 3 (SCL): 4_Zisterne(Fuellstand qm)

   // Füllstand Zisterne - An KNX rangieren
   "db-knx-ko".koVal."4_Zisterne(Fuellstand qm)" := "db-wasser".zisterne.fuellstand.qMeter;


   // 6/3/140 = Zisterne(Fuellstand qm)
   #"knx-KO"[4](Wert := "db-knx-ko".koVal."4_Zisterne(Fuellstand qm)",
                KNX_KO := "db-knx-ko".ko[4],
                KNX_Dat := "db-knx-com".KNXDat);
END_REGION

REGION Network 4 (SCL): 8_Zirkulation.WarmWasser(Ein)



   // 7/0/1 = Zirkulation.WarmWasser(Ein)
   #"knx-KO"[8](Wert := "db-knx-ko".koVal."8_Zirkulation.WarmWasser(Ein)",
                KNX_KO := "db-knx-ko".ko[8],
                KNX_Dat := "db-knx-com".KNXDat);
END_REGION

REGION Network 5 (SCL): 5_PV-Anlage(Erzeugung)
   (*
   Vom PV Anlage als W
   Auf dem KNX Bus als kW / DPT 9.024 Leistung (kW)
   *)


   "db-knx-ko".koVal."5_PV-Anlage(Erzeugung)" := ("db-haus".strom.pv_W / 1000.0);


   // 6/3/141 = PV-Anlage(Erzeugung)
   #"knx-KO"[5](Wert := "db-knx-ko".koVal."5_PV-Anlage(Erzeugung)",
                KNX_KO := "db-knx-ko".ko[5],
                KNX_Dat := "db-knx-com".KNXDat);
END_REGION

REGION Network 6 (SCL): 6_Stromzaehler(In-Out-Aktuell)
   (*
   Vom Volkszähler als W
   Auf dem KNX Bus als kW / DPT 9.024 Leistung (kW)
   *)

   "db-knx-ko".koVal."6_Stromzaehler(In-Out-Aktuell)" := ("db-haus".strom.netz_W/1000.0);

   // 6/0/0 = Strom(Aktuell)
   #"knx-KO"[6](Wert := "db-knx-ko".koVal."6_Stromzaehler(In-Out-Aktuell)",
                KNX_KO := "db-knx-ko".ko[6],
                KNX_Dat := "db-knx-com".KNXDat);
END_REGION

REGION Network 7 (SCL): 7_Strom(Eigenverbrauch)

   // DPT 9.024 Leistung (kW)

   "db-knx-ko".koVal."7_Strom(Eigenverbrauch)" := ("db-haus".strom.eigenverbrauch_W / 1000.0);


   //6/0/1 = Stromzaehler(Eigenverbrauch)
   #"knx-KO"[7](Wert := "db-knx-ko".koVal."7_Strom(Eigenverbrauch)",
                KNX_KO := "db-knx-ko".ko[7],
                KNX_Dat := "db-knx-com".KNXDat);
END_REGION

REGION Network 8 (SCL): Helligkeitswerte


   //6/3/0   = Umwelt.Wetterstation(Helligkeit O Messwert)
   #"knx-KO"[9](Wert := "db-knx-ko".koVal."9_Umwelt.Wetterstation(Helligkeit O Messwert)",
                KNX_KO := "db-knx-ko".ko[9],
                KNX_Dat := "db-knx-com".KNXDat);

   //6/3/17 = Umwelt.Wetterstation(Helligkeit S Messwert)
   #"knx-KO"[10](Wert := "db-knx-ko".koVal."10_Umwelt.Wetterstation(Helligkeit S Messwert)",
                KNX_KO := "db-knx-ko".ko[10],
                KNX_Dat := "db-knx-com".KNXDat);

   //6/3/34 = Umwelt.Wetterstation(Helligkeit W Messwert)
   #"knx-KO"[11](Wert := "db-knx-ko".koVal."11_Umwelt.Wetterstation(Helligkeit W Messwert)",
                KNX_KO := "db-knx-ko".ko[11],
                KNX_Dat := "db-knx-com".KNXDat);

   //6/3/105 = Umwelt-Garage.Lichtsensor(Helligkeit Messwert)
   #"knx-KO"[12](Wert := "db-knx-ko".koVal."12_Umwelt-Garage.Lichtsensor(Helligkeit Messwert)",
                KNX_KO := "db-knx-ko".ko[12],
                KNX_Dat := "db-knx-com".KNXDat);
END_REGION

REGION Network 9 (SCL): Beschattung(Diag)

   // 3/1/221 = Beschattung(Diag) 
   #"knx-KO"[13](Wert := "db-knx-ko".koVal."13_Beschattung(Diag)",
                KNX_KO := "db-knx-ko".ko[13],
                KNX_Dat := "db-knx-com".KNXDat);
END_REGION

REGION Network 10 (SCL): Wind Geschwindigkeit, Temperatur

   //6/3/54 = Umwelt.Wetterstation(Wind Geschwindigkeit)
   #"knx-KO"[14](Wert := "db-knx-ko".koVal."14_Umwelt.Wetterstation(Wind Geschwindigkeit)",
                 KNX_KO := "db-knx-ko".ko[14],
                 KNX_Dat := "db-knx-com".KNXDat);

   //6/3/55 = Umwelt.Wetterstation(Temperatur Messwert)
   #"knx-KO"[15](Wert := "db-knx-ko".koVal."15_Umwelt.Wetterstation(Temperatur Messwert)",
                 KNX_KO := "db-knx-ko".ko[15],
                 KNX_Dat := "db-knx-com".KNXDat);
END_REGION

REGION Network 11 (SCL): Helligkeit Maximal

   // 6/3/106 = Umwelt.Helligkeit.Max(Helligkeit)
   #"knx-KO"[16](Wert := "db-knx-ko".koVal."16_Umwelt.Helligkeit.Max(Helligkeit)",
                 KNX_KO := "db-knx-ko".ko[16],
                 KNX_Dat := "db-knx-com".KNXDat);
END_REGION

REGION Network 12 (SCL): Umwelt.Regensensor


   // 6/3/100 = Umwelt.Regensensor(Meldung Regen ja/nein)
   #"knx-KO"[17](Wert := "db-knx-ko".koVal."17_Umwelt.Regensensor(Meldung Regen ja/nein)",
                 KNX_KO := "db-knx-ko".ko[17],
                 KNX_Dat := "db-knx-com".KNXDat);
END_REGION

REGION Network 13 (SCL): 18_DPT3_Test

   // 11/0/10 = DPT3 Test
   #"knx-KO"[18](Wert := "db-knx-ko".koVal."18_DPT3_Test",
                 KNX_KO := "db-knx-ko".ko[18],
                 KNX_Dat := "db-knx-com".KNXDat);
END_REGION
END_FUNCTION_BLOCK

FUNCTION_BLOCK "knx-com"   // FB12, FBD
{ S7_Optimized_Access := 'TRUE' }
VERSION : 0.1
   VAR
      "knx-init-scan_Instance" : "knx-init-scan";
      fl_initscan1 : Bool;
      fl_initScan2 : Bool;
      "TON_knx<Bereit" : TON_TIME;
   END_VAR
   VAR_TEMP
      tmpGA : Word;
      tmpGaEq : Bool;
   END_VAR
   VAR_TEMP   // added for the SCL form of the ladder/FBD networks
      _w1 : Bool;
      _w2 : Bool;
   END_VAR
BEGIN

REGION Network 1: KNX Baustein
   // Zustände der Kommunikation!
   // 5:       Startverzögerungszeit läuft!
   // 10:     Eigene IP der SPS ermitteln! (RDREC-Baustein)
   // 12:     Initialisierung Tunnel-Status-Telegramm
   // 15:     Ethernet Verbindungsparameter initialisieren
   // 20:     Ethernet-Verbindung einrichten (TCON-Baustein)
   // 30:     Aufbau-Tunnel-Verbindung-Telegramm senden
   // 40:     Warte auf Bestätigung das der Tunnel aufgebaut ist!
   // 100:    Verbindung augebaut! Tunnel Telegramme können gesendet/empfangen werden
   // 110:    Lebenszeichen wird gesendet!
   // 115:    Lebenszeichen wurde von der Schnittstelle quittiert!
   // 120:    Verbindungsabbau-Anforderung erhalten! Verbindungsabbau bestätigen!
   // 150:    Tunneltelegramm erhalten! Bestätigung schicken
   // 200:    Tunneltelegramm schicken!
   // 210:    Warte auf Bestätigung der gesendeten Tunneldaten!
   // 250:    Tunnelverbindung soll abgebaut werden!
   // 260:    Tunnel abbauen! Warte auf Bestätigung!
   // 270:    Ethernet-Verbindung freigeben! (TDISON-Baustein)
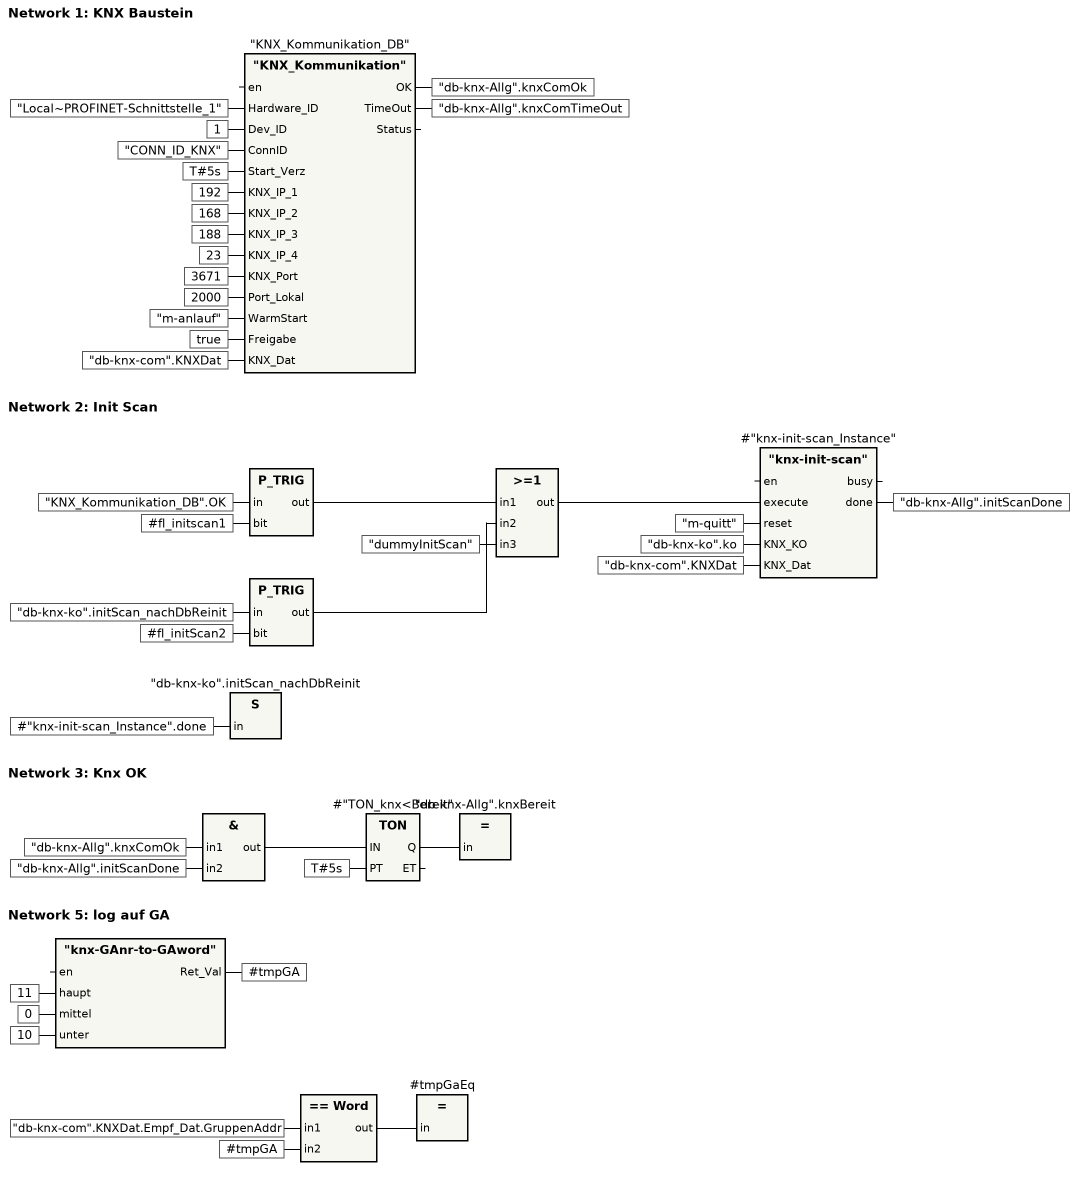
   "KNX_Kommunikation_DB"(Hardware_ID := "Local~PROFINET-Schnittstelle_1",   // "KNX_Kommunikation"
                          Dev_ID := 1,
                          ConnID := "CONN_ID_KNX",
                          Start_Verz := T#5s,
                          KNX_IP_1 := 192,
                          KNX_IP_2 := 168,
                          KNX_IP_3 := 188,
                          KNX_IP_4 := 23,
                          KNX_Port := 3671,
                          Port_Lokal := 2000,
                          WarmStart := "m-anlauf",
                          Freigabe := true,
                          KNX_Dat := "db-knx-com".KNXDat,
                          OK => "db-knx-Allg".knxComOk,
                          TimeOut => "db-knx-Allg".knxComTimeOut);
END_REGION

REGION Network 2: Init Scan
   // "dummyInitScan"
   #_w1 := "KNX_Kommunikation_DB".OK AND NOT #fl_initscan1;   // rising edge
   #fl_initscan1 := "KNX_Kommunikation_DB".OK;
   #_w2 := "db-knx-ko".initScan_nachDbReinit AND NOT #fl_initScan2;   // rising edge
   #fl_initScan2 := "db-knx-ko".initScan_nachDbReinit;
   #"knx-init-scan_Instance"(execute := #_w1 OR #_w2 OR "dummyInitScan",   // "knx-init-scan"
                           reset := "m-quitt",
                           KNX_KO := "db-knx-ko".ko,
                           KNX_Dat := "db-knx-com".KNXDat,
                           done => "db-knx-Allg".initScanDone);
   IF #"knx-init-scan_Instance".done THEN "db-knx-ko".initScan_nachDbReinit := TRUE; END_IF;
END_REGION

REGION Network 3: Knx OK
   #"TON_knx<Bereit"(IN := "db-knx-Allg".knxComOk AND "db-knx-Allg".initScanDone, PT := T#5s);   // TON
   "db-knx-Allg".knxBereit := #"TON_knx<Bereit".Q;
END_REGION

REGION Network 5: log auf GA
   // 11/0/10 = DPT3 Test
   #tmpGA := "knx-GAnr-to-GAword"(haupt := 11, mittel := 0, unter := 10);
   #tmpGaEq := "db-knx-com".KNXDat.Empf_Dat.GruppenAddr = #tmpGA;
END_REGION

REGION Network 6 (SCL): log


   IF "db-knx-com".KNXDat.Empfangen AND #tmpGaEq AND "m-knx-log-enable" THEN
       FOR "db-knx-log".index := 99 TO 0 BY -1 DO

           // umkopieren
           "db-knx-log".empf["db-knx-log".index + 1] := "db-knx-log".empf["db-knx-log".index];

           // neue daten sichern
           IF "db-knx-log".index = 0 THEN
               "db-knx-log".empf[0].Empf_Dat := "db-knx-com".KNXDat.Empf_Dat;
               "db-knx-log".empf[0].ga_nr := "knx-GAword-to-GAnr"("db-knx-log".empf[0].Empf_Dat.GruppenAddr);
           END_IF;

       END_FOR;
   END_IF;
END_REGION
END_FUNCTION_BLOCK

// folder: 20 KNX/KNX Bausteine

FUNCTION_BLOCK "knx-SendByChange"   // FB5, SCL
{ S7_Optimized_Access := 'TRUE' }
VERSION : 0.1
   VAR_INPUT
      wert : Variant;   // Wert der gesenden twerden soll
      aenderungWert : Real;   // Differen um die sich der Wert ändern muss damit er gesendet wird (Nur bei "Zahlen-Werte" relevant)
      sendenOk : Bool;   // Rückmeldung des KNX Bausteins
   END_VAR
   VAR_OUTPUT
      senden : Bool;   // Senden Trigger an KNX Baustein
   END_VAR
   VAR
      statSenden : Bool;
      statBoolAlt : Bool;
      statByteAlt : Byte;
      statWordAlt : Word;
      statIntAlt : Int;
      statUIntAlt : UInt;
      statRealAlt : Real;
   END_VAR
   VAR_TEMP
      tmp_Bool : Bool;
      tmp_Byte : Byte;
      tmp_sInt : SInt;
      tmp_usInt : USInt;
      tmp_Word : Word;
      tmp_Int : Int;
      tmp_UInt : UInt;
      tmp_Real : Real;
      tmp_diffInt : Int;
      tmp_diffUInt : UInt;
      tmp_diffReal : Real;
   END_VAR
BEGIN
   (*

   SendByChange

   Hilfsbaustein zum generieren eine Sende Triggers wenn sich der Wert in der SPS geändert hat

   17.10.2021 van
   Code aufgeräumt
   DPTs hinzugefügt

   09.2021 van
   Baustein erstellt und getestet

   *)


   // Senden Trigger zurücksetzen wenn senden erfolgreich war
   IF #sendenOk AND #statSenden THEN
       #statSenden := false;
   END_IF;


   // Wert auf Änderung überprüfen
   CASE TypeOf(#wert) OF

           // DPT 1   1 Bit   0..1 
           // 1.yyy = boolesch
       Bool:

           VariantGet(SRC := #wert,
                      DST => #tmp_Bool);

           IF #tmp_Bool <> #statBoolAlt THEN
               #statBoolAlt := #tmp_Bool;
               #statSenden := true;
           END_IF;


           //DPT 4   1 Byte, Char    1 ASCII-Zeichen Hinweis: Es sind nur ASCII-Zeichen ohne Steuerzeichen (mit Ausnahme von TAB, CR und LF) erlaubt.
           //DPT 5   1 Byte, Integer 0..255
           //DPT 6   1 Byte, Integer -128..127
           //4.yyy = Zeichen (8-Bit)
           //5.yyy = vorzeichenloser 8-Bit-#Wert, wie Dimm-#Wert (0..100 %), Jalousienposition (0..100 %)
           //6.yyy = 8-Bit-2-Komplement, z. B. %
       Byte:

           VariantGet(SRC := #wert,
                      DST => #tmp_Byte);


           IF #tmp_Byte <> #statByteAlt THEN
               #statByteAlt := #tmp_Byte;
               #statSenden := true;
           END_IF;


           //DPT 5   1 Byte, Integer 0..255
           //5.yyy = vorzeichenloser 8-Bit-#Wert, wie Dimm-#Wert (0..100 %), Jalousienposition (0..100 %)
       USInt:
           VariantGet(SRC := #wert,
                      DST => #tmp_usInt);

           #tmp_diffInt := ABS(#tmp_usInt - #statIntAlt);

           IF #tmp_diffInt >= REAL_TO_INT(#aenderungWert) THEN
               #statIntAlt := #tmp_Int;
               #statSenden := true;
           END_IF;


           //DPT 6   1 Byte, Integer -128..127
           //6.yyy = 8-Bit-2-Komplement, z. B. %
       SInt:
           VariantGet(SRC := #wert,
                      DST => #tmp_sInt);

           #tmp_diffInt := ABS(#tmp_sInt - #statIntAlt);

           IF #tmp_diffInt >= REAL_TO_INT(#aenderungWert) THEN
               #statIntAlt := #tmp_Int;
               #statSenden := true;
           END_IF;


           // DPT 7   2 Byte, Integer 0..65535    
           // DPT 8   2 Byte, Integer -32767..32767
           // DPT 9   2 Byte, Float   -671088,64..670760,96
           // 7.yyy = 2 x vorzeichenloser 8-Bit-Wert, z. B. Impulszähler
           // 8.yyy = 2 x 8-Bit-2-Komplement, z. B. %
       Word:
           VariantGet(SRC := #wert,
                      DST => #tmp_Word);

           IF #tmp_Word <> #statWordAlt THEN
               #statWordAlt := #tmp_Byte;
               #statSenden := true;
           END_IF;


           // DPT 7   2 Byte, Integer 0..65535
           // 7.yyy = 2 x vorzeichenloser 8-Bit-Wert, z. B. Impulszähler
       UInt:

           VariantGet(SRC := #wert,
                      DST => #tmp_UInt);

           #tmp_diffUInt := ABS(#tmp_UInt - #tmp_diffUInt);

           IF #tmp_diffInt >= REAL_TO_INT(#aenderungWert) THEN
               #statUIntAlt := #tmp_UInt;
               #statSenden := true;
           END_IF;


           // DPT 8   2 Byte, Integer -32767..32767    
           // 8.yyy = 2 x 8-Bit-2-Komplement, z. B. %
       Int:

           VariantGet(SRC := #wert,
                      DST => #tmp_Int);

           #tmp_diffInt := ABS(#tmp_Int - #statIntAlt);

           IF #tmp_diffInt >= REAL_TO_INT(#aenderungWert) THEN
               #statIntAlt := #tmp_Int;
               #statSenden := true;
           END_IF;


       Real:  //Gleitpunkt-Zahl  //DPT 9.xxx

           VariantGet(SRC := #wert,
                      DST => #tmp_Real);

           #tmp_diffReal := ABS(#tmp_Real - #statRealAlt);

           IF #tmp_diffReal >= #aenderungWert THEN
               #statRealAlt := #tmp_Real;
               #statSenden := true;
           END_IF;

       ELSE

           ;
   END_CASE;


   // Senden triggern
   #senden := #statSenden;
END_FUNCTION_BLOCK

FUNCTION_BLOCK "knx-init-scan"   // FB6, SCL
{ S7_Optimized_Access := 'TRUE' }
VERSION : 0.1
   VAR_INPUT
      execute : Bool;
      reset : Bool;
   END_VAR
   VAR_OUTPUT
      busy : Bool;
      done : Bool;
   END_VAR
   VAR_IN_OUT
      KNX_KO : Array[0.."KNX_ARRAY_MAX"] of "KNX_KO";
      KNX_Dat : "KNX_Data_Exchange";
   END_VAR
   VAR
      i : Int;
      R_TRIG_execute : R_TRIG;
      statSenden : Bool;
      statSendenOK : Bool;
      statBusy : Bool;
      statDone : Bool;
      "knx-txBus-GroupValueRead_Instance" : "knx-txBus-GroupValueRead";
   END_VAR
BEGIN
   (*

   knx-init-scan

   Der Baustein führt einen InitScan auf dem Bus durch

   Da beim Einschalten der SPS die relevanten KO-Werte in der SPS noch umbekannt sind.
   Dieser Baustein sendet beim Einschalten daher für alle entsprechend Parametrierten KOs 
   ein GroupValueRead auf den Bus.

   Folgende Parameter müssen true sein:
   "db-knx-ko".ko[x].para.aktiv
   "db-knx-ko".ko[x].para.beschreibbarVomBus
   "db-knx-ko".ko[x].para.initScan

   Und das KO muss in "knx-ko-aufrufe" entsprechend aufgerufen werden, damit der Wert zugewiesen werden kann.


   01.10.2022
   execute überarbeitet
   neu reset und busy

   17.10.2021 van
   Baustein erstellt

   *)

   //Start
   #R_TRIG_execute(CLK:=#execute);
   IF #R_TRIG_execute.Q THEN
       #i := 0;
       #statSenden := false;

       #statBusy := true;
       #statDone := false;
   END_IF;

   // Reset
   IF #reset THEN
       #statSenden := false;
       #statBusy := false;
       #statDone := false;
   END_IF;




   IF #statBusy AND (NOT #statDone) THEN

       // ReadRequest an den Bus senden ?
       IF #KNX_KO[#i].para.aktiv AND #KNX_KO[#i].para.initScan THEN
           #statSenden := true;
       ELSIF (NOT #KNX_KO[#i].para.aktiv) OR (NOT #KNX_KO[#i].para.initScan) THEN    // KO Init Scan nicht aktiv
           #statSenden := false;
           #i += 1;
       END_IF;

       // ReadRequest wurde an den Bus gesendet
       IF #statSenden AND #statSendenOK THEN
           #statSenden := false;
           #i += 1;
       END_IF;

   END_IF;



   // Fertig, Done
   IF #i > "KNX_ARRAY_MAX" THEN
       #statBusy := false;
       #statDone := true;
       #statSenden := false;
       #i := 0;
   END_IF;


   // ReadRequest Baustein
       #"knx-txBus-GroupValueRead_Instance"(haupt:=#KNX_KO[#i].GA.haupt,
                                        mittel:=#KNX_KO[#i].GA.mittel,
                                        unter:=#KNX_KO[#i].GA.unter,
                                        Senden:=#statSenden,
                                        Senden_OK=>#statSendenOK,
                                        KNX_Dat:=#KNX_Dat);


   // Out
   #busy := #statBusy;
   #done := #statDone;
END_FUNCTION_BLOCK

FUNCTION_BLOCK "knx-rxBus-GroupValueRead"   // FB7, SCL
{ S7_Optimized_Access := 'TRUE' }
VERSION : 0.1
   VAR_INPUT
      haupt : USInt;   // Hauptgruppe = 0..31
      mittel : USInt;   // Mittelgruppe = 0..7
      unter : USInt;   // Untergruppe = 0..255
   END_VAR
   VAR_OUTPUT
      GroupValueRead : Bool;
   END_VAR
   VAR_IN_OUT
      KNX_Dat : "KNX_Data_Exchange";
   END_VAR
   VAR
      GruppenAddr : Word;
   END_VAR
BEGIN
   (*

   knx-rxBus-GroupValueRead

   Hilfsbaustein um Leseanfrage vom Bus zu beantworten
   Der Baustein genereiert einen Trigger, wenn vom Bus eine Leseanfrage (GroupValueRead) auf die GA empfangen wird
   Der Trigger wird dann mit dem senden Eingang des KNX-Bausteins verbunden

   27.09.2021 van
   Baustein erstellt und getestet

   *)

   (*

   Daten[1] : Das Nutzdaten-Feld enthält eine Service-Kennung + die DATEN, 
   die von diesem Service verwendet werden sollen. Die Service-Kennung 
   wird als APCI bezeichnet, die Abkürzung für 
   Application Layer Protocol Control Information 
   (Anwendungsschicht-Protokoll-Kontrolldaten).

   ---------------

   Die APCI Daten sind auf ZWEI Bytes aufgeteil

         NPDU_ABCI        //        Daten[1]
                    /    APCI    / 6Bit Nutzdaten
   D8/D7/D6/D5/D4/D3/D2/D1//D8/D7/D6/D5/D4/D3/D2/D1

   ---------------

   GroupValueRead:     APCI = 0000b -> Daten[1] = 16#00
   GroupValueResponse: APCI = 0001b
   GroupValueWrite:    APCI = 0010b -> Daten[1] = 16#80

   ---------------

   https://support.knx.org/hc/de/articles/115003188529-Nutzdaten
   https://support.knx.org/hc/de/articles/115003189825-Telegrammtypen

   *)


   //Gruppenadresse zu einem Wort zusammenbauen!
   #GruppenAddr := "knx-GAnr-to-GAword"(haupt := #haupt, mittel := #mittel, unter := #unter);


   (*

   GroupValueRead Telegramm vom Bus empfangen wenn
    - Daten empfangen
    - GA stimmt
    - D8+D7 = 0, bzw einfachhalber Daten[1] = 0 , da keine Nutzdaten enthalten
      (GroupValueRead:     APCI = 0000b -> Daten[1] = 16#00)

   *)


   #GroupValueRead := #KNX_Dat.Empfangen AND (#KNX_Dat.Empf_Dat.GruppenAddr = #GruppenAddr) AND (#KNX_Dat.Empf_Dat.Daten[1] = 16#00);
END_FUNCTION_BLOCK

FUNCTION_BLOCK "knx-txBus-GroupValueRead"   // FB8, SCL
{ S7_Optimized_Access := 'TRUE' }
VERSION : 0.1
   VAR_INPUT
      haupt : USInt;   // Hauptgruppe = 0..31
      mittel : USInt;   // Mittelgruppe = 0..7
      unter : USInt;   // Untergruppe = 0..255
      Senden : Bool;
   END_VAR
   VAR_OUTPUT
      Senden_OK : Bool;   // Daten wurden auf den KNX-Bus übermittelt!
   END_VAR
   VAR_IN_OUT
      KNX_Dat : "KNX_Data_Exchange";
   END_VAR
   VAR
      GruppenAddr : Word;
      Gesendet : Bool;
      SendeAnf : Bool;
      R_TRIG_Senden : R_TRIG;
   END_VAR
BEGIN
   (*

   knx-txBus-GroupValueRead

   Hilfsbaustein um eine Leseanfrage (GroupValueRead) an den Bus zu senden
   Der Baustein sendet ein GroupValueRead an den Bus

   03.10.2021 van
   Baustein erstellt und getestet

   *)



   (*

   Daten[1] : Das Nutzdaten-Feld enthält eine Service-Kennung + die DATEN, 
   die von diesem Service verwendet werden sollen. Die Service-Kennung 
   wird als APCI bezeichnet, die Abkürzung für 
   Application Layer Protocol Control Information 
   (Anwendungsschicht-Protokoll-Kontrolldaten).

   ---------------

   Die APCI Daten sind auf ZWEI Bytes aufgeteil

         NPDU_ABCI        //        Daten[1]
                    /    APCI    / 6Bit Nutzdaten
   D8/D7/D6/D5/D4/D3/D2/D1//D8/D7/D6/D5/D4/D3/D2/D1

   ---------------

   GroupValueRead:     APCI = 0000b -> Daten[1] = 16#00
   GroupValueResponse: APCI = 0001b
   GroupValueWrite:    APCI = 0010b -> Daten[1] = 16#80

   ---------------

   https://support.knx.org/hc/de/articles/115003188529-Nutzdaten
   https://support.knx.org/hc/de/articles/115003189825-Telegrammtypen

   *)


   //Gruppenadresse zu einem Wort zusammenbauen!
   #GruppenAddr := "knx-GAnr-to-GAword"(haupt := #haupt, mittel := #mittel, unter := #unter);


   //Daten senden!
   #R_TRIG_Senden(CLK := #Senden);
   IF #R_TRIG_Senden.Q THEN
       #SendeAnf := true;   //Speichern, dass die Daten gesendet sollen!
   END_IF;


   IF #SendeAnf AND NOT #KNX_Dat.Senden THEN   //Nur wenn KNX_Daten.Senden "false" ist, können Daten gesendet werden!

       #KNX_Dat.Send_Dat.GruppenAddr := #GruppenAddr;
       #KNX_Dat.Send_Dat.Laenge := 16#01;

       // GroupValueRead:     APCI = 0000b -> Daten[1] = 16#00
       // Der einfachhalber können beide Byte Felder 0 sein, da es eh keine Daten gibt
       #KNX_Dat.Send_Dat.NPDU_ABCI := 16#00;
       #KNX_Dat.Send_Dat.Daten[1] := 16#00;

       #KNX_Dat.Senden := true;
       #SendeAnf := false;
       #Gesendet := true;

   END_IF;


   //Bit zurücksenden wenn der "Senden"-Input zurückgenommen wird!
   IF NOT #Senden THEN
       #Gesendet := false;
   END_IF;
   #Senden_OK := #Gesendet & NOT #KNX_Dat.Senden;
END_FUNCTION_BLOCK

FUNCTION_BLOCK "knx-sendenEmpfangen"   // FB9, SCL
{ S7_Optimized_Access := 'TRUE' }
VERSION : 0.1
   VAR_INPUT
      haupt : USInt;   // Hauptgruppe = 0..31
      mittel : USInt;   // Mittelgruppe = 0..7
      unter : USInt;   // Untergruppe = 0..255
      Senden : Bool;   // Sendet #Wert auf den Bus
      EmpfFrg : Bool;   // Gibt das beschreuben von #Wert VOM Bus frei
   END_VAR
   VAR_OUTPUT
      Senden_OK : Bool;   // Daten wurden auf den KNX-Bus übermittelt!
      Empf_OK : Bool;   // Daten wurden vom KNX-Bus empfangen!
   END_VAR
   VAR_IN_OUT
      Wert : Variant;   // Zu sendender / Empfangender Wert!
      KNX_Dat : "KNX_Data_Exchange";
   END_VAR
   VAR
      GruppenAddr : Word;
      Gesendet : Bool;
      SendeAnf : Bool;
      R_TRIG_Senden : R_TRIG;
      statAPCI : Byte;
   END_VAR
   VAR_TEMP
      tmp_bool : Bool;
      tmp_DPT3 : "KNX_DPT3";
      tmp_Byte : Byte;
      tmp_sInt : SInt;
      tmp_usInt : USInt;
      tmp_Word : Word;
      tmp_Int : Int;
      tmp_UInt : UInt;
      tmp_Dword : DWord;
      tmp_Real : Real;
      tmp_String : String [14];
      i : Int;
   END_VAR
BEGIN
   (*

   Der Baustein sendet bzw. empfängt ein KO vom Bus


   Die SPS Variable wird als Variant an #Wert übergeben
   Anhand des SPS-Datentyp wird das KNX-DPT "ermittelt"




   Quelle:
   "KNX_GruppeAddr" von kürbis85 und Matthias92
   https://www.sps-forum.de/threads/knx-kommunkation-%C3%BCber-knxnet-ip-mit-siemens-s7-1500-s7-1200-tia-portal.93641/

   20.02.2024 van
   DPT 3 implementiert

   02.06.2022 van
   Empfangen DPT 16 String ergänzt

   17.10.2021 van
   Code aufgeräumt
   DPTs hinzugefügt

   03.10.2021 van
   Baustein erstellt, auf Basic des Code von "KNX_GruppeAddr" von kürbis85 und Matthias92

   *)



   (*

   =========================
   DPT - Datenpunkttyp
   =========================


   Die am häufigsten verwendeten Datenpunkttypen sind:

   1.yyy = boolesch, wie Schalten, Bewegen nach oben/unten, Schritt
   2.yyy = 2 x boolesch, z. B. Schalten + Prioritätssteuerung
   3.yyy = boolesch + vorzeichenloser 3-Bit-Wert, z. B. Auf-/Abdimmen
   4.yyy = Zeichen (8-Bit)
   5.yyy = vorzeichenloser 8-Bit-Wert, wie Dimm-Wert (0..100 %), Jalousienposition (0..100 %)
   6.yyy = 8-Bit-2-Komplement, z. B. %
   7.yyy = 2 x vorzeichenloser 8-Bit-Wert, z. B. Impulszähler
   8.yyy = 2 x 8-Bit-2-Komplement, z. B. %
   9.yyy = 16-Bit-Gleitkommazahl, z. B. Temperatur
   10.yyy = Uhrzeit
   11.yyy = Datum
   12.yyy = 4 x vorzeichenloser 8-Bit-Wert,z. B. Impulszähler
   13.yyy = 4 x 8-Bit-2-Komplement, z. B. Impulszähler
   14.yyy = 32-Bit-Gleitkommazahl, z. B. Temperatur
   15.yyy = Zugangskontrolle
   16.yyy = String -> 14 Zeichen (14 x 8-Bit)
   17.yyy = Szenennummer
   18.yyy = Szenensteuerung
   19.yyy = Uhrzeit + Datum
   20.yyy = 8-Bit-Nummerierung,z. B. HLK-Modus („Automatik“, „Komfort“, „Stand-by“, „Sparen“, „Schutz“)

   https://support.knx.org/hc/de/articles/115001133744-Datenpunkttyp


   DPT 1   1 Bit   0..1    
   DPT 2   2 Bit   0..3    
   DPT 3   4 Bit   0..15   
   DPT 4   1 Byte, Char    1 ASCII-Zeichen Hinweis: Es sind nur ASCII-Zeichen ohne Steuerzeichen (mit Ausnahme von TAB, CR und LF) erlaubt.
   DPT 5   1 Byte, Integer 0..255  
   DPT 6   1 Byte, Integer -128..127   
   DPT 7   2 Byte, Integer 0..65535    
   DPT 8   2 Byte, Integer -32767..32767   
   DPT 9   2 Byte, Float   -671088,64..670760,96   
   DPT 10  3 Byte, Wochentag und Uhrzeit   "T.HH:MM:SS"    
   DPT 11  3 Byte, Datum   "JJJJ-MM-TT"    
   DPT 12  4 Byte, Integer 0..4294967295   
   DPT 13  4 Byte, Integer -2147483647..2147483647 
   DPT 14  4 Byte, Float   -∞..∞   Hinweis: Der Wertebereich hängt von der Anzahl der Nachkommastellen ab und ist daher nicht genau definierbar.
   DPT 16  14 Byte, String 14 ASCII-Zeichen


   *)




   //Gruppenadresse zu einem Wort zusammenbauen!
   #GruppenAddr := "knx-GAnr-to-GAword"(haupt := #haupt, mittel := #mittel, unter := #unter);


   REGION Senden zum Bus

       //Daten senden!
       #R_TRIG_Senden(CLK := #Senden);
       IF #R_TRIG_Senden.Q THEN
           #SendeAnf := true;   //Speichern, dass die Daten gesendet sollen!
       END_IF;

       IF #SendeAnf AND NOT #KNX_Dat.Senden THEN   //Nur wenn KNX_Daten.Senden "false" ist, können Daten gesendet werden!


           CASE TypeOf(#Wert) OF

                   // DPT 1   1 Bit   0..1 
                   // 1.yyy = boolesch
               Bool:
                   VariantGet(SRC := #Wert,
                              DST => #tmp_bool);

                   #KNX_Dat.Send_Dat.GruppenAddr := #GruppenAddr;
                   #KNX_Dat.Send_Dat.Laenge := 16#01;
                   #KNX_Dat.Send_Dat.NPDU_ABCI := 16#00;

                   IF #tmp_bool THEN
                       #KNX_Dat.Send_Dat.Daten[1] := 16#81;
                   ELSE
                       #KNX_Dat.Send_Dat.Daten[1] := 16#80;
                   END_IF;

                   #KNX_Dat.Senden := true;
                   #SendeAnf := false;
                   #Gesendet := true;


                // DPT 3   4 Bit   0..15     
                // 3.yyy = boolesch + vorzeichenloser 3-Bit-Wert, z. B. Auf-/Abdimmen   
               "KNX_DPT3":

                   VariantGet(SRC := #Wert,
                              DST => #tmp_DPT3);

                   #KNX_Dat.Send_Dat.GruppenAddr := #GruppenAddr;
                   #KNX_Dat.Send_Dat.Laenge := 16#01;
                   #KNX_Dat.Send_Dat.NPDU_ABCI := 16#00;

                   #tmp_Byte := "knx-plc-to-DPT3"(#tmp_DPT3);

                   #KNX_Dat.Send_Dat.Daten[1] := #tmp_Byte;
                   #KNX_Dat.Send_Dat.Daten[1].%X7 := true; // 16#8x

                   #KNX_Dat.Senden := true;
                   #SendeAnf := false;
                   #Gesendet := true;



                   //DPT 4   1 Byte, Char    1 ASCII-Zeichen Hinweis: Es sind nur ASCII-Zeichen ohne Steuerzeichen (mit Ausnahme von TAB, CR und LF) erlaubt.
                   //DPT 5   1 Byte, Integer 0..255
                   //DPT 6   1 Byte, Integer -128..127
                   //4.yyy = Zeichen (8-Bit)
                   //5.yyy = vorzeichenloser 8-Bit-#Wert, wie Dimm-#Wert (0..100 %), Jalousienposition (0..100 %)
                   //6.yyy = 8-Bit-2-Komplement, z. B. %
               Byte:
                   VariantGet(SRC := #Wert,
                              DST => #tmp_Byte);
                   #KNX_Dat.Send_Dat.GruppenAddr := #GruppenAddr;
                   #KNX_Dat.Send_Dat.Laenge := 16#02;
                   #KNX_Dat.Send_Dat.NPDU_ABCI := 16#00;

                   #KNX_Dat.Send_Dat.Daten[1] := 16#80;
                   #KNX_Dat.Send_Dat.Daten[2] := #tmp_Byte;

                   #KNX_Dat.Senden := true;
                   #SendeAnf := false;
                   #Gesendet := true;


                   //DPT 5   1 Byte, Integer 0..255
                   //5.yyy = vorzeichenloser 8-Bit-#Wert, wie Dimm-#Wert (0..100 %), Jalousienposition (0..100 %)
               USInt:
                   VariantGet(SRC := #Wert,
                              DST => #tmp_usInt);
                   #KNX_Dat.Send_Dat.GruppenAddr := #GruppenAddr;
                   #KNX_Dat.Send_Dat.Laenge := 16#02;
                   #KNX_Dat.Send_Dat.NPDU_ABCI := 16#00;

                   #KNX_Dat.Send_Dat.Daten[1] := 16#80;
                   #KNX_Dat.Send_Dat.Daten[2] := USINT_TO_BYTE(#tmp_usInt);

                   #KNX_Dat.Senden := true;
                   #SendeAnf := false;
                   #Gesendet := true;


                   //DPT 6   1 Byte, Integer -128..127
                   //6.yyy = 8-Bit-2-Komplement, z. B. %
               SInt:
                   VariantGet(SRC := #Wert,
                              DST => #tmp_sInt);
                   #KNX_Dat.Send_Dat.GruppenAddr := #GruppenAddr;
                   #KNX_Dat.Send_Dat.Laenge := 16#02;
                   #KNX_Dat.Send_Dat.NPDU_ABCI := 16#00;

                   #KNX_Dat.Send_Dat.Daten[1] := 16#80;
                   #KNX_Dat.Send_Dat.Daten[2] := SINT_TO_BYTE(#tmp_sInt);

                   #KNX_Dat.Senden := true;
                   #SendeAnf := false;
                   #Gesendet := true;


                   // DPT 7   2 Byte, Integer 0..65535    
                   // DPT 8   2 Byte, Integer -32767..32767
                   // DPT 9   2 Byte, Float   -671088,64..670760,96
                   // 7.yyy = 2 x vorzeichenloser 8-Bit-Wert, z. B. Impulszähler
                   // 8.yyy = 2 x 8-Bit-2-Komplement, z. B. %
               Word:
                   VariantGet(SRC := #Wert,
                              DST => #tmp_Word);
                   #KNX_Dat.Send_Dat.GruppenAddr := #GruppenAddr;
                   #KNX_Dat.Send_Dat.Laenge := 16#03;
                   #KNX_Dat.Send_Dat.NPDU_ABCI := 16#00;

                   #KNX_Dat.Send_Dat.Daten[1] := 16#80;
                   #KNX_Dat.Send_Dat.Daten[2] := #tmp_Word.%B1;
                   #KNX_Dat.Send_Dat.Daten[3] := #tmp_Word.%B0;

                   #KNX_Dat.Senden := true;
                   #SendeAnf := false;
                   #Gesendet := true;


                   // DPT 7   2 Byte, Integer 0..65535    
                   // 7.yyy = 2 x vorzeichenloser 8-Bit-Wert, z. B. Impulszähler
               UInt:
                   VariantGet(SRC := #Wert,
                              DST => #tmp_UInt);

                   #KNX_Dat.Send_Dat.GruppenAddr := #GruppenAddr;
                   #KNX_Dat.Send_Dat.Laenge := 16#03;
                   #KNX_Dat.Send_Dat.NPDU_ABCI := 16#00;

                   #KNX_Dat.Send_Dat.Daten[1] := 16#80;
                   #KNX_Dat.Send_Dat.Daten[2] := #tmp_UInt.%B1;
                   #KNX_Dat.Send_Dat.Daten[3] := #tmp_UInt.%B0;

                   #KNX_Dat.Senden := true;
                   #SendeAnf := false;
                   #Gesendet := true;


                   // DPT 8   2 Byte, Integer -32767..32767    
                   // 8.yyy = 2 x 8-Bit-2-Komplement, z. B. %
               Int:
                   VariantGet(SRC := #Wert,
                              DST => #tmp_Int);

                   #KNX_Dat.Send_Dat.GruppenAddr := #GruppenAddr;
                   #KNX_Dat.Send_Dat.Laenge := 16#03;
                   #KNX_Dat.Send_Dat.NPDU_ABCI := 16#00;

                   #KNX_Dat.Send_Dat.Daten[1] := 16#80;
                   #KNX_Dat.Send_Dat.Daten[2] := #tmp_Int.%B1;
                   #KNX_Dat.Send_Dat.Daten[3] := #tmp_Int.%B0;

                   #KNX_Dat.Senden := true;
                   #SendeAnf := false;


                   //9.yyy = 16-Bit-Gleitkommazahl, z. B. Temperatur  
               Real:
                   VariantGet(SRC := #Wert,
                              DST => #tmp_Real);
                   #KNX_Dat.Send_Dat.GruppenAddr := #GruppenAddr;
                   #KNX_Dat.Send_Dat.Laenge := 16#03;
                   #KNX_Dat.Send_Dat.NPDU_ABCI := 16#00;


                   #tmp_Word := "knx-real-to-DPT9"(#tmp_Real);

                   #KNX_Dat.Send_Dat.Daten[1] := 16#80;
                   #KNX_Dat.Send_Dat.Daten[2] := #tmp_Word.%B1;
                   #KNX_Dat.Send_Dat.Daten[3] := #tmp_Word.%B0;

                   #KNX_Dat.Senden := true;
                   #SendeAnf := false;
                   #Gesendet := true;


                   //String   //DPT 16.xxx 
                   //16.yyy = String -> 14 Zeichen (14 x 8-Bit)
               String:
                   VariantGet(SRC := #Wert,
                              DST => #tmp_String);
                   #KNX_Dat.Send_Dat.GruppenAddr := #GruppenAddr;
                   #KNX_Dat.Send_Dat.Laenge := 16#0F;
                   #KNX_Dat.Send_Dat.NPDU_ABCI := 16#00;
                   #KNX_Dat.Send_Dat.Daten[1] := 16#80;
                   #KNX_Dat.Send_Dat.Daten[2] := #tmp_String[1];
                   #KNX_Dat.Send_Dat.Daten[3] := #tmp_String[2];
                   #KNX_Dat.Send_Dat.Daten[4] := #tmp_String[3];
                   #KNX_Dat.Send_Dat.Daten[5] := #tmp_String[4];
                   #KNX_Dat.Send_Dat.Daten[6] := #tmp_String[5];
                   #KNX_Dat.Send_Dat.Daten[7] := #tmp_String[6];
                   #KNX_Dat.Send_Dat.Daten[8] := #tmp_String[7];
                   #KNX_Dat.Send_Dat.Daten[9] := #tmp_String[8];
                   #KNX_Dat.Send_Dat.Daten[10] := #tmp_String[9];
                   #KNX_Dat.Send_Dat.Daten[11] := #tmp_String[10];
                   #KNX_Dat.Send_Dat.Daten[12] := #tmp_String[11];
                   #KNX_Dat.Send_Dat.Daten[13] := #tmp_String[12];
                   #KNX_Dat.Send_Dat.Daten[14] := #tmp_String[13];
                   #KNX_Dat.Send_Dat.Daten[15] := #tmp_String[14];
                   #KNX_Dat.Senden := true;
                   #SendeAnf := false;
                   #Gesendet := true;


               ELSE  // Statement section ELSE
                   ;
           END_CASE;

       END_IF;
       //Bit zurücksenden wenn der "Senden"-Input zurückgenommen wird!
       IF NOT #Senden THEN
           #Gesendet := false;
       END_IF;
       #Senden_OK := #Gesendet & NOT #KNX_Dat.Senden;



   END_REGION


   REGION Empfangen vom Bus

       #Empf_OK := false;

       //APCI extrahieren
       // GroupValueRead:     APCI = 0000b 
       // GroupValueResponse: APCI = 0001b
       // GroupValueWrite:    APCI = 0010b 
       #statAPCI.%X3 := #KNX_Dat.Empf_Dat.NPDU_ABCI.%X1;
       #statAPCI.%X2 := #KNX_Dat.Empf_Dat.NPDU_ABCI.%X0;
       #statAPCI.%X1 := #KNX_Dat.Empf_Dat.Daten[1].%X7;
       #statAPCI.%X0 := #KNX_Dat.Empf_Dat.Daten[1].%X6;


       IF #KNX_Dat.Empfangen
           AND #EmpfFrg
           AND (#KNX_Dat.Empf_Dat.GruppenAddr = #GruppenAddr)
           AND ((#statAPCI = 2#0000_0001) OR (#statAPCI = 2#0000_0010))    //Auf beides reagieren: GroupValueResponse oder GroupValueWrite
       THEN

           CASE TypeOf(#Wert) OF

                   // 1.yyy = boolesch
               Bool:
                   IF (#KNX_Dat.Empf_Dat.Laenge = 16#01)
                   THEN
                       #KNX_Dat.Empfangen := false;

                       // Daten aufbereiten
                       #tmp_bool := #KNX_Dat.Empf_Dat.Daten[1].%X0;
                       VariantPut(SRC := #tmp_bool,
                                  DST := #Wert);

                       #Empf_OK := TRUE;
                   END_IF;


                   // DPT 3   4 Bit   0..15     
                   // 3.yyy = boolesch + vorzeichenloser 3-Bit-Wert, z. B. Auf-/Abdimmen   
               "KNX_DPT3":
                   IF (#KNX_Dat.Empf_Dat.Laenge = 16#01)
                   THEN
                       #KNX_Dat.Empfangen := false;

                       // Daten aufbereiten
                       #tmp_DPT3:="knx-DPT3-to-plc"(data:=#KNX_Dat.Empf_Dat.Daten[1]);

                       VariantPut(SRC := #tmp_DPT3,
                                  DST := #Wert);

                       #Empf_OK := TRUE;
                   END_IF;



                   //DPT 4   1 Byte, Char    1 ASCII-Zeichen Hinweis: Es sind nur ASCII-Zeichen ohne Steuerzeichen (mit Ausnahme von TAB, CR und LF) erlaubt.
                   //DPT 5   1 Byte, Integer 0..255
                   //DPT 6   1 Byte, Integer -128..127
                   //4.yyy = Zeichen (8-Bit)
                   //5.yyy = vorzeichenloser 8-Bit-#Wert, wie Dimm-#Wert (0..100 %), Jalousienposition (0..100 %)
                   //6.yyy = 8-Bit-2-Komplement, z. B. %
               Byte:
                   IF (#KNX_Dat.Empf_Dat.Laenge = 16#02)
                   THEN
                       #KNX_Dat.Empfangen := false;

                       // Daten aufbereiten
                       #tmp_Byte := #KNX_Dat.Empf_Dat.Daten[2];

                       VariantPut(SRC := #tmp_Byte,
                                  DST := #Wert);

                       #Empf_OK := TRUE;
                   END_IF;


                   //DPT 5   1 Byte, Integer 0..255
                   //5.yyy = vorzeichenloser 8-Bit-#Wert, wie Dimm-#Wert (0..100 %), Jalousienposition (0..100 %)
               SInt:
                   IF (#KNX_Dat.Empf_Dat.Laenge = 16#02)
                   THEN
                       #KNX_Dat.Empfangen := false;

                       // Daten aufbereiten
                       #tmp_sInt := BYTE_TO_SINT(#KNX_Dat.Empf_Dat.Daten[2]);
                       VariantPut(SRC := #tmp_sInt,
                                  DST := #Wert);

                       #Empf_OK := TRUE;
                   END_IF;


                   //DPT 6   1 Byte, Integer -128..127
                   //6.yyy = 8-Bit-2-Komplement, z. B. %  
               USInt:
                   IF (#KNX_Dat.Empf_Dat.Laenge = 16#02)
                   THEN
                       #KNX_Dat.Empfangen := false;

                       // Daten aufbereiten
                       #tmp_usInt := BYTE_TO_USINT(#KNX_Dat.Empf_Dat.Daten[2]);
                       VariantPut(SRC := #tmp_usInt,
                                  DST := #Wert);

                       #Empf_OK := TRUE;
                   END_IF;


                   // DPT 7   2 Byte, Integer 0..65535    
                   // DPT 8   2 Byte, Integer -32767..32767
                   // DPT 9   2 Byte, Float   -671088,64..670760,96
                   // 7.yyy = 2 x vorzeichenloser 8-Bit-Wert, z. B. Impulszähler
                   // 8.yyy = 2 x 8-Bit-2-Komplement, z. B. %
               Word:
                   IF (#KNX_Dat.Empf_Dat.Laenge = 16#03)
                   THEN
                       #KNX_Dat.Empfangen := false;

                       // Daten aufbereiten
                       #tmp_Word.%B1 := #KNX_Dat.Empf_Dat.Daten[2];
                       #tmp_Word.%B0 := #KNX_Dat.Empf_Dat.Daten[3];
                       VariantPut(SRC := #tmp_Word,
                                  DST := #Wert);

                       #Empf_OK := TRUE;
                   END_IF;


                   // DPT 7   2 Byte, Integer 0..65535    
                   // 7.yyy = 2 x vorzeichenloser 8-Bit-Wert, z. B. Impulszähler
               UInt:
                   IF (#KNX_Dat.Empf_Dat.Laenge = 16#03)
                   THEN
                       #KNX_Dat.Empfangen := false;

                       // Daten aufbereiten
                       #tmp_Int.%B1 := #KNX_Dat.Empf_Dat.Daten[2];
                       #tmp_Int.%B0 := #KNX_Dat.Empf_Dat.Daten[3];
                       VariantPut(SRC := #tmp_UInt,
                                  DST := #Wert);

                       #Empf_OK := TRUE;
                   END_IF;


                   // DPT 8   2 Byte, Integer -32767..32767    
                   // 8.yyy = 2 x 8-Bit-2-Komplement, z. B. %  
               Int:
                   IF (#KNX_Dat.Empf_Dat.Laenge = 16#03)
                   THEN
                       #KNX_Dat.Empfangen := false;

                       // Daten aufbereiten
                       #tmp_Int.%B1 := #KNX_Dat.Empf_Dat.Daten[2];
                       #tmp_Int.%B0 := #KNX_Dat.Empf_Dat.Daten[3];
                       VariantPut(SRC := #tmp_Int,
                                  DST := #Wert);

                       #Empf_OK := TRUE;
                   END_IF;


                   //9.yyy = 16-Bit-Gleitkommazahl, z. B. Temperatur
               Real:
                   IF (#KNX_Dat.Empf_Dat.Laenge = 16#03)
                   THEN
                       #KNX_Dat.Empfangen := false;


                       // Daten aufbereiten
                       #tmp_Word.%B0 := #KNX_Dat.Empf_Dat.Daten[3];
                       #tmp_Word.%B1 := #KNX_Dat.Empf_Dat.Daten[2];
                       #tmp_Real := "knx-DPT9-to-real"(#tmp_Word);

                       VariantPut(SRC := #tmp_Real,
                                  DST := #Wert);

                       #Empf_OK := TRUE;
                   END_IF;


                // DPT 16  14 Byte, String 14 ASCII-Zeichen
                // 16.yyy = String -> 14 Zeichen (14 x 8-Bit)
               String:
                   IF (#KNX_Dat.Empf_Dat.Laenge = 16#0F)
                   THEN
                       #KNX_Dat.Empfangen := false;

                       // Daten aufbereiten
                       // erstes Zeichen in #KNX_Dat.Empf_Dat.Daten[2]

                       #tmp_String := '              ';    // String init

                       FOR #i := 1 TO 14 DO
                           IF #KNX_Dat.Empf_Dat.Daten[#i + 1] <> 0 THEN
                               #tmp_String[#i] := #KNX_Dat.Empf_Dat.Daten[#i + 1];
                           ELSE
                               #tmp_String[#i] := ' ';
                           END_IF;

                       END_FOR;

                       VariantPut(SRC := #tmp_String,
                                  DST := #Wert);

                       #Empf_OK := TRUE;
                   END_IF;

               ELSE  // Statement section ELSE
                   ;
           END_CASE;
       END_IF;


   END_REGION
END_FUNCTION_BLOCK

FUNCTION_BLOCK "KNX_Kommunikation"   // FB11, SCL
{ S7_Optimized_Access := 'TRUE' }
VERSION : 0.1
   VAR_INPUT
      Hardware_ID : Hw_Io := 16#64;   // Hardwarekennung der Ethernetschnittstelle!
      Dev_ID : Byte;   // 1= Lokale PN-Schnittstelle!
      ConnID : Word;   // Verknüpfung der SEND und RCV-Bausteine; Eindeutige Abstimmung CPU weit!
      Start_Verz : Time;   // Startverzögerung bei einem Neustart der CPU! KNX-Schnittstelle Zeit zum hochfahren geben!
      KNX_IP_1 : Byte;   // IP-Adresse der KNX Schnittstelle! Teil 1 Bsp."192"
      KNX_IP_2 : Byte;   // IP-Adresse der KNX Schnittstelle! Teil 2 Bsp."168"
      KNX_IP_3 : Byte;   // IP-Adresse der KNX Schnittstelle! Teil 3 Bsp."1"
      KNX_IP_4 : Byte;   // IP-Adresse der KNX Schnittstelle! Teil 4 Bsp."100"
      KNX_Port : UInt;   // Zugriffsport der KNX-Schnittstelle!
      Port_Lokal : UInt;   // Lokaler Port der SPS!
      WarmStart : Bool;   // Flanke CPU wurde neugestartet!
      Freigabe : Bool;   // Verbindung / Kommunikation soll aufgebaut werden!
   END_VAR
   VAR_OUTPUT
      OK : Bool;   // Kommunikation wurde augebaut!
      TimeOut : Bool;   // Keine Antwort von der KNX-Schnittstelle!
      Status : Int;   // Aktueller Zustand der Kommunikation!
   END_VAR
   VAR_IN_OUT
      KNX_Dat : "KNX_Data_Exchange";
   END_VAR
   VAR
      R_TRIG_Aufbauen : R_TRIG;
      RDREC_Instance : RDREC;
      PDInterfaceDataReal : Struct
         BlockType : UInt;
         BlockLength : UInt;
         BlockVersionHigh : USInt;
         BlockVersionLow : USInt;
         Data : Array[0..301] of Byte;
         OwnChassisID : String;
      END_STRUCT;
      STATUS_RDEC : DWord;   // Fehlerrückgabe RDREC-Baustein! (Eigene IP einlesen)
      STATUS_TCON : Word;   // Fehlerrückgabe TCON-Baustein!
      STATUS_URCV : Word;   // Fehlerrückgabe URCV-Baustein!
      STATUS_USEND : Word;   // Fehlerrückgabe USEND-Baustein!
      STATUS_TDISCON : Word;   // Fehlerrückgabe TDISCON-Baustein!
      R_TRIG_URCV_NDR : R_TRIG;
      F_TRIG_Senden : F_TRIG;
      IEC_Timer_Lebenszeichen : TON_TIME;
      IEC_Timer_TimeOut : TON_TIME;
      ETH_Connect_Para : TCON_Param;
      KNX_Endpunkt : TADDR_Param;
      TCON : TCON;
      USEND : TUSEND;
      URCV : TURCV;
      TDISCON : TDISCON;
      EigeneIP : Array[1..4] of Byte;
      RcvData : Array[1..100] of Byte;
      SendData : Array[1..100] of Byte;
      KNX : Struct
         ChannelID : Byte;
         Addr : Word;
         ConnectionType : Byte;   // Sollte eine 4 sein laug Beispiel!
         "Counter" : Byte;
         SeqNrSenden : Byte;
         SeqNrEmpf : Byte;
      END_STRUCT;
      KNXInfo : Struct   // Rein Informativ zur Fehlerfindung!
         ServiceType0208_ErrorCode : Byte;
         ServiceType0206_ErrorCode : Byte;
         SendeTicks : DInt;   // Anzahl gesendeter Telegramme
         EmpfTicks : DInt;   // Anzahl Empfangs-Telegramme
         Typ206Ticks : DInt;   // Anzahl Empfangs-Telegramme
         Typ208Ticks : DInt;   // Anzahl Empfangs-Telegramme
         Typ209Ticks : DInt;   // Anzahl Empfangs-Telegramme
         Typ20ATicks : DInt;   // Anzahl Empfangs-Telegramme
         Typ420Ticks : DInt;   // Anzahl Empfangs-Telegramme
         Typ421Ticks : DInt;   // Anzahl Empfangs-Telegramme
      END_STRUCT;
      EmpfServ : Struct
         Type206_Ok : Bool;   // Tunnel aufbau erhalten!
         Type206_Err : Bool;   // Tunnel aufbau erhalten! Error
         Type208_OK : Bool;   // Lebenstelegramm antwort erhalten!
         Type208_Err : Bool;   // Lebenstelegramm antwort erhalten! Nicht OK
         Type209_Da : Bool;   // Diconnect Anforderung erhalten
         Type20A_OK : Bool;   // Verbindungsabbau wurde bestätigt!
         Type420_Da : Bool;   // Bus-Telegramm erhalten!
         Type421_OK : Bool;   // Bus-Telegramm wurde bestätigt!
      END_STRUCT;
      T : Struct
         AnfTunnel : Struct
            IP_Header : Struct
               HeaderSize : Byte;
               ProtokollVersion : Byte;
               ServiceType : Word;
               TotalLaenge : Word;
            END_STRUCT;
            IP_Body : Struct
               HPAI_Control_Endpoint : Struct
                  Laenge : Byte;
                  ProtocolCode : Byte;
                  IP1 : Byte;
                  IP2 : Byte;
                  IP3 : Byte;
                  IP4 : Byte;
                  Port : Word;
               END_STRUCT;
               HPAI_Data_EndPoint : Struct
                  Laenge : Byte;
                  ProtocolCode : Byte;
                  IP1 : Byte;
                  IP2 : Byte;
                  IP3 : Byte;
                  IP4 : Byte;
                  Port : Word;
               END_STRUCT;
               CRI : Struct   // Connection Request Information
                  Laenge : Byte;
                  ConnectionTypCode : Byte;
                  KNX_Layer : Byte;
                  Reserve : Byte;
               END_STRUCT;
            END_STRUCT;
         END_STRUCT;
         AnfTunnelACK : Struct
            IP_Header : Struct
               HeaderSize : Byte;
               ProtokollVersion : Byte;
               ServiceType : Word;
               TotalLaenge : Word;
            END_STRUCT;
            IP_Body : Struct
               CummunicationChannel : Byte;
               StatusCode : Byte;
               Data_EndPoint : Struct
                  Laenge : Byte;
                  ProtocolCode : Byte;
                  IP1 : Byte;
                  IP2 : Byte;
                  IP3 : Byte;
                  IP4 : Byte;
                  Port : Word;
               END_STRUCT;
               CRD : Struct
                  Laenge : Byte;
                  ConnectionTypCode : Byte;
                  InidviduelleAddr : Word;
               END_STRUCT;
            END_STRUCT;
         END_STRUCT;
         AnfTunnelState : Struct
            IP_Header : Struct
               HeaderSize : Byte;
               ProtokollVersion : Byte;
               ServiceType : Word;
               TotalLaenge : Word;
            END_STRUCT;
            IP_Body : Struct
               CummunicationChannel : Byte;
               Reserve : Byte;
               Control_EndPoint : Struct
                  Laenge : Byte;
                  ProtocolCode : Byte;
                  IP1 : Byte;
                  IP2 : Byte;
                  IP3 : Byte;
                  IP4 : Byte;
                  Port : Word;
               END_STRUCT;
            END_STRUCT;
         END_STRUCT;
         AnfTunnelStateACK : Struct
            IP_Header : Struct
               HeaderSize : Byte;
               ProtokollVersion : Byte;
               ServiceType : Word;
               TotalLaenge : Word;
            END_STRUCT;
            IP_Body : Struct
               CummunicationChannel : Byte;
               Statuscode : Byte;
            END_STRUCT;
         END_STRUCT;
         Tunnel : Struct
            IP_Header : Struct
               HeaderSize : Byte;
               ProtokollVersion : Byte;
               ServiceType : Word;
               TotalLaenge : Word;
            END_STRUCT;
            Conn_Header : Struct
               Laenge : Byte;
               ChannelID : Byte;
               SequenzeCount : Byte;
               Reserve : Byte;
            END_STRUCT;
            Cemi : Struct
               MessageCode : Byte;
               AdditionalLaenge : Byte;
               Kontrollbyte1 : Byte;
               Kontrollbyte2 : Byte;
               SourceAddr : Word;
               DestinationAddr : Word;
            END_STRUCT;
            NPDU : Struct
               Laenge : Byte;
               NPDU_ABCI : Byte;
               Daten : Array[1..20] of Byte;
            END_STRUCT;
         END_STRUCT;
         TunnelAck : Struct
            IP_Header : Struct
               HeaderSize : Byte;
               ProtokollVersion : Byte;
               ServiceType : Word;
               TotalLaenge : Word;
            END_STRUCT;
            IP_Body : Struct
               Laenge : Byte;
               ChannelID : Byte;
               SequenzCount : Byte;
               Status : Byte;
            END_STRUCT;
         END_STRUCT;
      END_STRUCT;
      SendeLaenge : DInt;
      State : Int;   // Aktueller Zustand der Kommunikation!
      SendeAnf : Int;   // 1=TunnelREQ, 2=Lebenszeichen, 3=Disconnect, 4=TunnelTeleACK, 5=Daten senden
      RueckState : Int;   // Ruecksprung Status
      ServiceType : Word;   // Empfangender Servicetype
      Senden : Bool;   // Ein Telegram soll verschickt werden!
      SendeFrg : Bool;   // EinTelegramm darf verschickt werden!
      DatenDa : Bool;   // Ein neues Telegramm wurde empfangen!
      HMTimeOut : Bool;
      IEC_Timer_StartVerz : TON_TIME;
   END_VAR
   VAR_TEMP
      POS : DInt;
      fehler : Int;
      i : Int;
      DummyUSInt : USInt;
      DummyInt : Int;
   END_VAR
BEGIN
   ////////////////////////////////////////////////////////////////////////////////////////////
   //                                                                                        
   //                                  BUSTEIN INFORMATIONEN                                 
   //                                                                                                                         
   //  Version:        1.0                                                                   
   //  Ersteller:      Brand                                                                 
   //  Titel:          KNX_Kommunikation                                        
   //  Erstelldatum:   2018                                                            
   //                                                                                        
   // Dieser Baustein kommuniziert über die Ethernet-Schnittstelle mit einer KNX-Bus-Schnittstelle!
   // 
   // ÄNDERUNGEN:
   // V1.0    2018   Erstinbetriebnahme
   //  
   // 
   ////////////////////////////////////////////////////////////////////////////////////////////
   (*  Zustände der Kommunikation!
   5:      Startverzögerungszeit läuft!
   10:     Eigene IP der SPS ermitteln! (RDREC-Baustein)
   12:     Initialisierung Tunnel-Status-Telegramm
   15:     Ethernet Verbindungsparameter initialisieren
   20:     Ethernet-Verbindung einrichten (TCON-Baustein)
   30:     Aufbau-Tunnel-Verbindung-Telegramm senden
   40:     Warte auf Bestätigung das der Tunnel aufgebaut ist!
   100:    Verbindung augebaut! Tunnel Telegramme können gesendet/empfangen werden
   110:    Lebenszeichen wird gesendet!
   115:    Lebenszeichen wurde von der Schnittstelle quittiert!
   120:    Verbindungsabbau-Anforderung erhalten! Verbindungsabbau bestätigen!
   150:    Tunneltelegramm erhalten! Bestätigung schicken
   200:    Tunneltelegramm schicken!
   210:    Warte auf Bestätigung der gesendeten Tunneldaten!
   250:    Tunnelverbindung soll abgebaut werden!
   260:    Tunnel abbauen! Warte auf Bestätigung!
   270:    Ethernet-Verbindung freigeben! (TDISON-Baustein)    
   *)

   #R_TRIG_Aufbauen(CLK := #Freigabe);
   //Kommunikation starten!
   IF (#WarmStart & #Freigabe) OR #R_TRIG_Aufbauen.Q THEN
       #State:=5;
   END_IF;

   #KNX_Dat.Empfangen := false;

   //Empfangsaufruf
   #URCV(EN_R := #State >= 30 AND NOT #DatenDa,
         ID := #ConnID,
               LEN := 0,
               DATA := #RcvData,
               ADDR := #KNX_Endpunkt);
         #R_TRIG_URCV_NDR(CLK := #URCV.NDR);
   IF  #R_TRIG_URCV_NDR.Q THEN
             #DatenDa := true;
             #KNXInfo.EmpfTicks := #KNXInfo.EmpfTicks + 1;
             #STATUS_URCV := 0;
             #ServiceType := #RcvData[3];
             #ServiceType :=SHL(IN:=#ServiceType , N:=8)OR #RcvData[4] ;
         END_IF;
   IF #URCV.ERROR THEN
             #STATUS_URCV := #URCV.STATUS;
         END_IF;

   IF #DatenDa THEN
             //Tunnelaufbau Bestätigung
             IF #ServiceType = 16#0206 THEN
                 IF #EmpfServ.Type206_Ok = false AND #EmpfServ.Type206_Err = false THEN
                     #KNXInfo.Typ206Ticks := #KNXInfo.Typ206Ticks + 1;
                     #DatenDa := false;
                     #fehler := Deserialize(SRC_ARRAY := #RcvData, DEST_VARIABLE => #T.AnfTunnelACK, POS := #POS);
                     IF #fehler = 0 THEN
                         IF #T.AnfTunnelACK.IP_Body.StatusCode = 0 THEN
                             IF #T.AnfTunnelACK.IP_Body.Data_EndPoint.IP1 = #KNX_IP_1 &
                                 #T.AnfTunnelACK.IP_Body.Data_EndPoint.IP2 = #KNX_IP_2 &
                                 #T.AnfTunnelACK.IP_Body.Data_EndPoint.IP3 = #KNX_IP_3 &
                                 #T.AnfTunnelACK.IP_Body.Data_EndPoint.IP4 = #KNX_IP_4 &
                                 #T.AnfTunnelACK.IP_Body.Data_EndPoint."Port" = #KNX_Port
                             THEN
                                 #KNX.ChannelID := #T.AnfTunnelACK.IP_Body.CummunicationChannel;
                                 #KNX.Addr := #T.AnfTunnelACK.IP_Body.CRD.InidviduelleAddr;
                                 #KNX.ConnectionType := #T.AnfTunnelACK.IP_Body.CRD.ConnectionTypCode;
                                 #KNX.Counter := #KNX.Counter + 1;
                                 #EmpfServ.Type206_Ok := true;
                             END_IF;
                         ELSE
                             #KNXInfo.ServiceType0206_ErrorCode := #T.AnfTunnelACK.IP_Body.StatusCode;
                             #EmpfServ.Type206_Err := true;
                         END_IF;
                     END_IF;
                 END_IF;
             END_IF;
             //Lebenstelegramm erhalten    
             IF #ServiceType = 16#208 THEN
                 IF #EmpfServ.Type208_OK = false AND #EmpfServ.Type208_Err = FALSE THEN
                     #KNXInfo.Typ208Ticks := #KNXInfo.Typ208Ticks + 1;
                     #DatenDa := false;
                     #fehler := Deserialize(SRC_ARRAY := #RcvData, DEST_VARIABLE => #T.AnfTunnelStateACK, POS := #POS);
                     IF #fehler = 0 THEN
                         IF #T.AnfTunnelStateACK.IP_Body.Statuscode = 0 THEN
                             IF #T.AnfTunnelStateACK.IP_Body.CummunicationChannel = #KNX.ChannelID THEN
                                 #KNXInfo.ServiceType0208_ErrorCode := 0;
                                 #EmpfServ.Type208_OK := true;
                             END_IF;
                         ELSE
                             #KNXInfo.ServiceType0208_ErrorCode := #T.AnfTunnelStateACK.IP_Body.Statuscode;
                             #EmpfServ.Type208_Err := true;
                         END_IF;
                     END_IF;
                 END_IF;
             END_IF;
             //Disconnect Anforderung erhalten!
             IF #ServiceType = 16#209 THEN
                 IF #EmpfServ.Type209_Da = false THEN
                     #KNXInfo.Typ209Ticks := #KNXInfo.Typ209Ticks + 1;
                     #DatenDa := false;
                     #EmpfServ.Type209_Da := true;

                     #POS := 0;
                     #fehler := Deserialize(SRC_ARRAY := #RcvData, DEST_VARIABLE => #T.AnfTunnelState, POS := #POS);
                     IF #fehler = 0 THEN
                         IF #T.AnfTunnelState.IP_Body.Control_EndPoint.IP1 = #KNX_IP_1 &
                             #T.AnfTunnelState.IP_Body.Control_EndPoint.IP2 = #KNX_IP_2 &
                             #T.AnfTunnelState.IP_Body.Control_EndPoint.IP3 = #KNX_IP_3 &
                             #T.AnfTunnelState.IP_Body.Control_EndPoint.IP4 = #KNX_IP_4 &
                             #T.AnfTunnelState.IP_Body.Control_EndPoint."Port" = #KNX_Port
                         THEN
                             "db-knx-Allg"."Disconnect Count" := "db-knx-Allg"."Disconnect Count" + 1;
                             IF "db-knx-Allg"."Disconnect Count" >= 1 AND "db-knx-Allg"."Disconnect Count" <= 20 THEN
                                 "db-knx-Allg".DisconnectChannelID["db-knx-Allg"."Disconnect Count"] := #T.AnfTunnelState.IP_Body.CummunicationChannel;
                             END_IF;
                         END_IF;
                     END_IF;
                 END_IF;
             END_IF;
             //Verbindungsabbau Bestätigung erhalten!
             IF #ServiceType = 16#20A THEN
                 IF #EmpfServ.Type20A_OK = false THEN
                     #KNXInfo.Typ20ATicks := #KNXInfo.Typ20ATicks + 1;
                     #EmpfServ.Type20A_OK := true;
                   #DatenDa := false;
                 END_IF;
             END_IF;
             //Tunneltelegramm erhalten!
             IF #ServiceType = 16#420 THEN
                IF #EmpfServ.Type420_Da = false THEN
                    #KNXInfo.Typ420Ticks := #KNXInfo.Typ420Ticks + 1;
                    #EmpfServ.Type420_Da := true;
                    #DatenDa := false;
                    #POS := 0;
                    #fehler := Deserialize(SRC_ARRAY := #RcvData, DEST_VARIABLE => #T.Tunnel, POS := #POS);
                    #KNX.SeqNrEmpf := #T.Tunnel.Conn_Header.SequenzeCount;
                    #KNX_Dat.Empf_Dat.GruppenAddr := #T.Tunnel.Cemi.DestinationAddr;
                    #KNX_Dat.Empf_Dat.Laenge := #T.Tunnel.NPDU.Laenge;
                    #KNX_Dat.Empf_Dat.NPDU_ABCI := #T.Tunnel.NPDU.NPDU_ABCI;
                    #KNX_Dat.Empf_Dat.Daten := #T.Tunnel.NPDU.Daten;

                    #KNX_Dat.Empfangen := true;

                 END_IF;
             END_IF;
             //Gesendetes Tunneltelegramm bestätigt!
             IF #ServiceType = 16#421 THEN
                 IF #EmpfServ.Type421_OK = false THEN
                     #KNXInfo.Typ421Ticks := #KNXInfo.Typ421Ticks + 1;
                     #EmpfServ.Type421_OK := true;
                     #DatenDa := false;
                     #POS := 0;
                     #fehler := Deserialize(SRC_ARRAY := #RcvData, DEST_VARIABLE => #T.Tunnel, POS := #POS);
                     //#KNX.SeqNrEmpf := #T.Tunnel.Conn_Header.SequenzeCount;
                 END_IF;
             END_IF;
   END_IF;

   //Bit erzeugen; ob der Sendebaustein bereit ist für neue Aufträge!
   #F_TRIG_Senden(CLK:=#Senden);
   #SendeFrg := NOT #Senden AND NOT #F_TRIG_Senden.Q;


   //Zeiteinheiten
   #IEC_Timer_Lebenszeichen.TON(IN := #State >= 100 AND #State <> 110,
                                 PT := t#50s);
   #IEC_Timer_TimeOut.TON(IN:=#State=40 OR #State = 115 OR #State = 210 OR #State =260 ,
                           PT:=t#5s );

   //Bausteinaufrufe zur Initialisierung
   IF #State < 40 THEN
       #RDREC_Instance(REQ := #State = 10,
                       ID := #Hardware_ID,
                       INDEX := w#16#8080,
                       MLEN := 300,
                       RECORD := #PDInterfaceDataReal); //Eigene IP einlesen
       #TCON(REQ := #State = 20,
             ID := #ETH_Connect_Para.ID,
             CONNECT := #ETH_Connect_Para);
       #IEC_Timer_StartVerz(IN:=NOT #WarmStart,
                            PT:=#Start_Verz);
   END_IF;
   //Bausteinaufrufe Verbindung beenden!
   IF #State >= 250 THEN
       #TDISCON(REQ := #State = 270,
                       ID := #ConnID);
   END_IF;

   //Organisation der Kommunikation
   CASE #State OF
       5: //Startverzögerung; KNX-Schnittstelle Zeit zum hochfahren geben!
           IF #IEC_Timer_StartVerz.Q THEN
               #State := 10;
           END_IF;
       10:  // Eigene IP einlesen!
           IF #RDREC_Instance.ERROR THEN
               #STATUS_RDEC := #RDREC_Instance.STATUS;
           END_IF;
           IF #RDREC_Instance.VALID THEN
               #DummyUSInt := #PDInterfaceDataReal.Data[0] + (4 - ((#PDInterfaceDataReal.Data[0] + 2) MOD 4));
               #EigeneIP[1] := #PDInterfaceDataReal.Data[#DummyUSInt + 8 + 0];
               #EigeneIP[2] := #PDInterfaceDataReal.Data[#DummyUSInt + 8 + 1];
               #EigeneIP[3] := #PDInterfaceDataReal.Data[#DummyUSInt + 8 + 2];
               #EigeneIP[4] := #PDInterfaceDataReal.Data[#DummyUSInt + 8 + 3];
               #STATUS_RDEC := 0;
               #State := 12;
           END_IF;
       12: //Tunnel Status Telegramm initialisieren!
           #T.AnfTunnelState.IP_Header.HeaderSize := 16#06;
           #T.AnfTunnelState.IP_Header.ProtokollVersion := 16#10;
           #T.AnfTunnelState.IP_Header.ServiceType := 16#0207;
           #T.AnfTunnelState.IP_Header.TotalLaenge := 16#0010;

           #T.AnfTunnelState.IP_Body.Control_EndPoint.Laenge := 16#08;
           #T.AnfTunnelState.IP_Body.Control_EndPoint.ProtocolCode := 16#01;
           #T.AnfTunnelState.IP_Body.Control_EndPoint.IP1 := #EigeneIP[1];
           #T.AnfTunnelState.IP_Body.Control_EndPoint.IP2 := #EigeneIP[2];
           #T.AnfTunnelState.IP_Body.Control_EndPoint.IP3 := #EigeneIP[3];
           #T.AnfTunnelState.IP_Body.Control_EndPoint.IP4 := #EigeneIP[4];
           #T.AnfTunnelState.IP_Body.Control_EndPoint."Port" := #Port_Lokal;
           #State := 15;

       15: //Ethernet-Parameter initialisieren!
           #Senden := false;
           #DatenDa := false;
           //Verbindung Parametrieren
           #ETH_Connect_Para.BLOCK_LENGTH := 64;
           #ETH_Connect_Para.LOCAL_DEVICE_ID := #Dev_ID;
           // Verbindungs ID Muss auf der Steuerung einmalig sein
           #ETH_Connect_Para.ID := #ConnID;
           // 19 für eine UDP "Verbindung"
           #ETH_Connect_Para.CONNECTION_TYPE := 19;
           // Länge der Lokalen verbindungsParameter angeben. Bei UDP wird nur der Port benötigt somit 2 Byte
           #ETH_Connect_Para.LOCAL_TSAP_ID_LEN := 2;
           //Höherwertiges Byte des Ports eintragen
           #ETH_Connect_Para.LOCAL_TSAP_ID[1] := UINT_TO_BYTE(SHR(IN := #Port_Lokal, N := 8));
           //Niederwertiges Byte des Ports eintragen
           #ETH_Connect_Para.LOCAL_TSAP_ID[2] := UINT_TO_BYTE(#Port_Lokal);;
           //Aktiververbindungsaufbau auf false setzen. Achtung bei Tia ist diser bei der Datenstruktur standardmässig auf True bei Step7 ist er false !! 
           #ETH_Connect_Para.ACTIVE_EST := false;

           //Zieladresse zuweisen
           #KNX_Endpunkt.REM_IP_ADDR[1] := #KNX_IP_1;
           #KNX_Endpunkt.REM_IP_ADDR[2] := #KNX_IP_2;
           #KNX_Endpunkt.REM_IP_ADDR[3] := #KNX_IP_3;
           #KNX_Endpunkt.REM_IP_ADDR[4] := #KNX_IP_4;
           #KNX_Endpunkt.REM_PORT_NR := #KNX_Port;
           #KNX.Counter := 0;
           #State := 20;

       20: //Ethernet-Verbindung einrichten!
           // Port öffnen
            IF #TCON.ERROR THEN
               #STATUS_TCON := #TCON.STATUS;
           END_IF;

           //Port Geöffnet
           IF #TCON.DONE OR #TCON.STATUS = 16#80a3 THEN
               #STATUS_TCON := 0;
               #State := 30;
           END_IF;

       30: // KNX Tunnel aufbauen
           IF #SendeFrg THEN
               #SendeAnf := 1;
               #EmpfServ.Type206_Ok := false;
               #EmpfServ.Type206_Err := False;
               #KNX.ChannelID := 0;
               #State := 40;
           END_IF;

       40: //Warte auf Bestätigung das der Tunnel augebaut wurde!
           IF #EmpfServ.Type206_Ok THEN
               #EmpfServ.Type206_Ok := false;
               #State := 100;
               #KNX.SeqNrSenden := 0;

           END_IF;
           IF #EmpfServ.Type206_Err THEN
               #EmpfServ.Type206_Err := false;

               // #State := 10;
           END_IF;
           IF #EmpfServ.Type209_Da THEN   //Verbindungs-Abbau bestätigen!
               #State := 120;
               #RueckState := 40; 
           END_IF;
           IF #IEC_Timer_TimeOut.Q THEN   //Bei Time-Out neustart!
               #State := 10;
           END_IF;

       100: //Die Verbidnung steht, was soll gemacht werden?
           IF  #EmpfServ.Type209_Da THEN               //Verbindgsabbau Anforderung erhalten! Sofort bestätigen!
               #State := 120;
           ELSIF #EmpfServ.Type420_Da THEN             //Tunneltelegramm erhalten! Sofort bestätigen!
               #State := 150;
           ELSIF #IEC_Timer_Lebenszeichen.Q THEN       //Lebenstelegramm schicken! 
               #State := 110;
           ELSIF NOT #Freigabe  THEN                   //Kommunikation beenden!
               #State := 250;
               #RueckState := 0;
           ELSIF #KNX_Dat.Senden THEN                 //Tunneltelegramm senden!
               #State := 200;
           END_IF;


       110: //Lebenszeichen senden!
           IF #SendeFrg THEN
               #SendeAnf := 2;
               #State := 115;
           END_IF;

       115: //Lebenzeichen zurück gekommen?
           IF #EmpfServ.Type208_OK   THEN
               #EmpfServ.Type208_OK := false;
               #State := 100;

           END_IF;
           IF #EmpfServ.Type208_Err THEN
               ; #EmpfServ.Type208_Err := false;
               ;// #State := 100;
           END_IF;
           IF #EmpfServ.Type209_Da THEN   //Bei einem Verbindungsabbau-Telegramm dieses bestätigen!
               #RueckState := 115;
               #State := 120;
           END_IF;
           IF #IEC_Timer_TimeOut.Q THEN   //Bei Time-Out neustart!
               #State := 250;      //Verbindung beenden
               #RueckState := 10;  //anschließender Neustart!
           END_IF;
       120: // DISCONNECT Anforderung erhalten!
           IF #SendeFrg THEN
               #SendeAnf := 3;

               #EmpfServ.Type209_Da := false;
                IF #T.AnfTunnelState.IP_Body.CummunicationChannel = #KNX.ChannelID THEN
                    #State := 10;    //Aktuelle Verbindung soll abgebaut werden! Also Neustart!
                ELSE
                    IF #RueckState = 0 THEN
                        #State := 100;    //Nicht "unsere" Verbndung soll abgebaut werden! => Weitermachen    
                    ELSE
                        #State := #RueckState;
                    END_IF;
                END_IF;
           END_IF;
        150: //Empfangenes Tunneltelegramm antworten!
           IF #SendeFrg THEN
               #EmpfServ.Type420_Da := false;
               #SendeAnf := 4;
               #State := 100;
           END_IF;
       200: //Tunnel-Telegramm senden!
           IF #SendeFrg THEN
               #EmpfServ.Type421_OK := false;
               #SendeAnf := 5;
               #State := 210;
           END_IF;
       210: //Tunnel-Telegramm senden; Bestätigung erhalten?
           IF #EmpfServ.Type421_OK THEN
              #EmpfServ.Type421_OK := false;
               #KNX.SeqNrSenden := #KNX.SeqNrSenden + 1;

               #State := 100;
               #KNX_Dat.Senden := false;

           END_IF;
           IF #IEC_Timer_TimeOut.Q THEN   //Bei Time-Out neustart!
               #State := 250;      //Verbindung beenden
               #RueckState := 10;  //anschließender Neustart!
           END_IF;
       250: //Verbindungsabbau anfordern!
           IF #SendeFrg THEN
               #EmpfServ.Type20A_OK := false;
               #SendeAnf := 6;
               #State := 260;
           END_IF;
       260: //Verbindungsabbau anfordern; Bestätigung erhalten?
           IF #EmpfServ.Type20A_OK THEN
               #EmpfServ.Type20A_OK := false;
               #State := 270;
           END_IF;
           IF #IEC_Timer_TimeOut.Q THEN
               #State := 270;
           END_IF;
       270: //Ethernet-Verbidnung freigeben!
           IF #TDISCON.DONE OR #TDISCON.STATUS=16#80A3 THEN
               IF #RueckState = 0 THEN
                   #State := 0;
               ELSE
                   #State := #RueckState; //Neustart der Kommunikation!
               END_IF;
           END_IF;
           IF #TDISCON.ERROR THEN
               #STATUS_TDISCON := #TDISCON.STATUS;
               IF #RueckState = 0 THEN
                   #State := 0;
               ELSE
                   #State := #RueckState; //Neustart der Kommunikation!
               END_IF;
           END_IF;
   END_CASE;

   //Sendedaten aufbereiten!
   CASE #SendeAnf OF
           1://Tunnel Aufbauen!
               //Siehe KNX Spezifikation Kap.8.8.5!
                   #T.AnfTunnel.IP_Header.HeaderSize := 16#6;
                   #T.AnfTunnel.IP_Header.ProtokollVersion := 16#10;
                   #T.AnfTunnel.IP_Header.ServiceType := 16#0205;
                   #T.AnfTunnel.IP_Header.TotalLaenge := 16#001A; //16#1A => 26

                   #T.AnfTunnel.IP_Body.HPAI_Control_Endpoint.Laenge := 16#08;
                   #T.AnfTunnel.IP_Body.HPAI_Control_Endpoint.ProtocolCode := 16#01;  //=> 2049
                   #T.AnfTunnel.IP_Body.HPAI_Control_Endpoint.IP1 := #EigeneIP[1];
                   #T.AnfTunnel.IP_Body.HPAI_Control_Endpoint.IP2 := #EigeneIP[2];
                   #T.AnfTunnel.IP_Body.HPAI_Control_Endpoint.IP3 := #EigeneIP[3];
                   #T.AnfTunnel.IP_Body.HPAI_Control_Endpoint.IP4 := #EigeneIP[4];
                   #T.AnfTunnel.IP_Body.HPAI_Control_Endpoint."Port" := #Port_Lokal; //16#07D0;

                   #T.AnfTunnel.IP_Body.HPAI_Data_EndPoint.Laenge := 16#08;
                   #T.AnfTunnel.IP_Body.HPAI_Data_EndPoint.ProtocolCode := 16#01;
                   #T.AnfTunnel.IP_Body.HPAI_Data_EndPoint.IP1 := #EigeneIP[1];
                   #T.AnfTunnel.IP_Body.HPAI_Data_EndPoint.IP2 := #EigeneIP[2];
                   #T.AnfTunnel.IP_Body.HPAI_Data_EndPoint.IP3 := #EigeneIP[3];
                   #T.AnfTunnel.IP_Body.HPAI_Data_EndPoint.IP4 := #EigeneIP[4];
                   #T.AnfTunnel.IP_Body.HPAI_Data_EndPoint."Port" := #Port_Lokal; //16#07D0 => 2000;

                   #T.AnfTunnel.IP_Body.CRI.Laenge := 16#04;
                   #T.AnfTunnel.IP_Body.CRI.ConnectionTypCode := 16#04;
                   #T.AnfTunnel.IP_Body.CRI.KNX_Layer := 16#02;
                   #T.AnfTunnel.IP_Body.CRI.Reserve := 16#00;

                   #POS := 0;
                   #fehler := Serialize(SRC_VARIABLE := #T.AnfTunnel, DEST_ARRAY => #SendData, POS := #POS);

                   #SendeLaenge := #POS;
                   #Senden := true;

           2: //Lebenszeichen senden!
                       #T.AnfTunnelState.IP_Body.CummunicationChannel := INT_TO_BYTE(#KNX.ChannelID);
                       #POS := 0;
                       #fehler := Serialize(SRC_VARIABLE := #T.AnfTunnelState, DEST_ARRAY => #SendData, POS := #POS);

                       #SendeLaenge := #POS;
                       #Senden := true;

            3: //DISCONNECT Bestätigung senden!
                       #T.AnfTunnelStateACK.IP_Header.HeaderSize := 16#06;
                       #T.AnfTunnelStateACK.IP_Header.ProtokollVersion := 16#01;
                       #T.AnfTunnelStateACK.IP_Header.ServiceType := 16#020A;
                       #T.AnfTunnelStateACK.IP_Header.TotalLaenge := 16#08;

                       #T.AnfTunnelStateACK.IP_Body.CummunicationChannel :=#KNX.ChannelID;
                       #T.AnfTunnelStateACK.IP_Body.Statuscode := 16#00;

                       #POS := 0;
                       #fehler := Serialize(SRC_VARIABLE := #T.AnfTunnelStateACK, DEST_ARRAY => #SendData, POS := #POS);

                       #SendeLaenge := #POS;
                       #Senden := true;

                   4: //Tunneltelegramm bestätigen!
                       #EmpfServ.Type420_Da := false;

